// HIGH-PV - Hold if the silo level is too high
IF maxPVEnable AND autoMode THEN
    tonMaxPTrip   (IN := (whiteWaterSiloLevel > maxPVTripEng),       PT := maxPVTripTime);
    tonMaxPRelease(IN := (whiteWaterSiloLevel < maxPVReleaseEng),    PT := maxPVReleaseTime);
    IF tonMaxPTrip.Q    THEN maxPVHoldActive := TRUE;  END_IF;
    IF tonMaxPRelease.Q THEN maxPVHoldActive := FALSE; END_IF;

ELSE
    tonMaxPTrip(IN := FALSE);
    tonMaxPRelease(IN := FALSE);
    maxPVHoldActive := FALSE;
END_IF;

// ============================ PV HOLD aggregation ============================
// NOTE: Requires pvHoldActive : BOOL in VAR section
pvHoldActive := FALSE;
IF autoMode THEN
    pvHoldActive := (minPVEnable AND minPVHoldActive) OR
                    (maxPVEnable AND maxPVHoldActive);
END_IF;


// ============================ Immediate stop / safety/fault =================
IF rStop OR stopCommand THEN
    controlOutputPct := 0.0;
    running := FALSE;
    deviceState := 'Stopping (Stop command)';
    runLatch := FALSE;
    step := 90;
END_IF;

IF vfdFaultFeedback THEN
    deviceState := 'Fault from drive';
    runLatch := FALSE;
    step := 90;
END_IF;

IF NOT allSafetyOK THEN
    deviceState := 'Stopping: safety chain open';
    runLatch := FALSE;
    step := 90;
END_IF;


// ============================ State machine =====================
CASE step OF
    // ------------------------------------------------------------
    0: // Idle
        running := FALSE;
        controlOutputPct := 0.0;
        deviceState := 'Idle';
        vfdStartCmdOut := FALSE;

        // Start request via runLatch (toggled by Start pulse)
        IF runLatch AND NOT stopCommand THEN
            // Safety must be OK; drive must be ready
            // PV hold does NOT block start anymore; it will only inhibit reference to 0%
            IF NOT allSafetyOK THEN
                deviceState := 'Start blocked: safety not OK';
                runLatch := FALSE;
                step := 0;

            ELSIF NOT vfdReady THEN
                deviceState := 'Start blocked: drive not ready';
                runLatch := FALSE;
                step := 0;

            ELSE
                IF pvHoldActive THEN
                    deviceState := 'Starting (PV hold active: output inhibited)';
                ELSE
                    deviceState := 'Starting';
                END_IF;

                vfdStartCmdOut := TRUE;                   // send START to drive
                tonRunFbWait(IN := TRUE, PT := vfdRunFbTimeout);
                step := 10;
            END_IF
        END_IF

    // ------------------------------------------------------------
    10: // Starting (await RUN feedback)
        running := FALSE;
        deviceState := 'Starting (await RUN feedback)';
        vfdStartCmdOut := TRUE;

        // If PV hold is active during start, ensure reference is inhibited to 0%
        IF pvHoldActive THEN
            controlOutputPct := 0.0;
        END_IF;

        // Safety/fault during start => stop
        IF NOT allSafetyOK THEN
            tonRunFbWait(IN := FALSE);
            deviceState := 'Stopping: safety chain open';
            vfdStartCmdOut := FALSE;
            runLatch := FALSE;
            step := 90;

        ELSIF vfdFaultFeedback THEN
            tonRunFbWait(IN := FALSE);
            deviceState := 'Fault from drive';
            vfdStartCmdOut := FALSE;
            runLatch := FALSE;
            step := 90;

        // Interlocks are normal stop only
        ELSIF anyInterlockOpen THEN
            tonRunFbWait(IN := FALSE);
            deviceState := 'Stopping: interlock open';
            vfdStartCmdOut := FALSE;
            runLatch := FALSE;
            step := 90;

        // RUN feedback arrived
        ELSIF vfdRunFeedback THEN
            tonRunFbWait(IN := FALSE);
            step := 20;

        // Timeout
        ELSIF tonRunFbWait.Q THEN
            tonRunFbWait(IN := FALSE);
            deviceState := 'Start failed: RUN feedback timeout';
            vfdStartCmdOut := FALSE;
            runLatch := FALSE;
            step := 90;
        END_IF

    // ------------------------------------------------------------
    20: // Running (control loop)
        running := TRUE;               // may be used to release other devices
        deviceState := 'Running';
        vfdStartCmdOut := TRUE;

        // Supervision
        IF NOT allSafetyOK THEN
            deviceState := 'Stopping: safety chain open';
            vfdStartCmdOut := FALSE;
            runLatch := FALSE;
            step := 90;

        ELSIF vfdFaultFeedback THEN
            deviceState := 'Fault from drive';
            vfdStartCmdOut := FALSE;
            runLatch := FALSE;
            step := 90;

        ELSIF NOT vfdReady THEN
            deviceState := 'Stopping: drive not ready';
            vfdStartCmdOut := FALSE;
            runLatch := FALSE;
            step := 90;

        ELSIF NOT vfdRunFeedback THEN
            deviceState := 'Stopping: RUN feedback lost';
            vfdStartCmdOut := FALSE;
            runLatch := FALSE;
            step := 90;

        // Interlocks → normal stop
        ELSIF anyInterlockOpen THEN
            deviceState := 'Stopping: interlock open';
            vfdStartCmdOut := FALSE;
            runLatch := FALSE;
            step := 90;

        // Start toggled OFF while running => stop
        ELSIF NOT runLatch THEN
            deviceState := 'Stopping (Start toggled off)';
            vfdStartCmdOut := FALSE;
            step := 90;

        ELSE
            // ---- Input filtering (PT1) ----
            IF enableInputFilter THEN
                instPT1(in := whiteWaterSiloLevel, T := inputFilterTime, K := inputFilterGainK, out => pvEngFiltered);
            ELSE
                pvEngFiltered := whiteWaterSiloLevel;
            END_IF

            // ---- Engineering → % scaling ----
            IF enableScaling THEN
                pvPct := _ScaleToPct(pvEngFiltered,       pLoEng, pHiEng);
                spPct := _ScaleToPct(processSetpointAuto, pLoEng, pHiEng);
            ELSE
                pvPct := pvEngFiltered;        // already %
                spPct := processSetpointAuto;  // already %
            END_IF

            // ---- Manual path (HMI) ----
            manualCmd := LIMIT(0.0, processSetpointMan, 100.0);

            // Reverse/direct action by Kp sign
            IF reverseActing THEN
                kpUse := -ABS(kp);
            ELSE
                kpUse :=  ABS(kp);
            END_IF

            // ===================== PV HOLD behavior =====================
            // When PV hold active: keep motor energized, force reference=0.0,
            // and hold PID (avoid error/windup) by forcing SET=ACT and MAN=TRUE.
            IF pvHoldActive THEN

                deviceState := 'Running (PV hold: output inhibited)';
                vfdStartCmdOut := TRUE;        // keep energized
                running := TRUE;               // keep permissives (change to FALSE if you prefer)

                instPID(
                    ACT := pvPct,
                    SET := pvPct,              // hold: SET follows PV -> DIFF ~ 0
                    M_I := 0.0,                // forced output during hold
                    MAN := TRUE,               // hold PID
                    RST := resetPID,
                    KP  := kpUse,
                    TN  := tn,
                    TV  := tv,
//                    LL  := outLowLimitPct,
//                    LH  := outHighLimitPct,
                    Y   => yPID,
                    DIFF=> pidDiff,
                    LIM => pidLimited
                );

                // Output inhibited to zero, motor stays enabled
                controlOutputPct := 0.0;

            ELSE
                // ===================== Normal control =====================
                instPID(
                    ACT := pvPct,
                    SET := spPct,
                    M_I := manualCmd,
                    MAN := NOT autoMode,
                    RST := resetPID,
                    KP  := kpUse,
                    TN  := tn,
                    TV  := tv,
//                    LL  := outLowLimitPct,
//                    LH  := outHighLimitPct,
                    Y   => yPID,
                    DIFF=> pidDiff,
                    LIM => pidLimited
                );

                // Mode select, offset, clamp
                IF autoMode THEN
                    controlOutputPct := yPID;
					instPID.LL := outLowLimitPct;
					instPID.LH := outHighLimitPct;
				
					
                ELSE
                    controlOutputPct := manualCmd;
					instPID.LL := manualCmd;
					instPID.LH := manualCmd;
				
                END_IF

                controlOutputPct := LIMIT(outLowLimitPct, controlOutputPct + outputOffsetPct, outHighLimitPct);
            END_IF
        END_IF

    // ------------------------------------------------------------
    90: // Stopping (normal, de-energize)
        running := FALSE;
        controlOutputPct := 0.0;
        vfdStartCmdOut := FALSE;
        tonRunFbWait(IN := FALSE);

        // Return to Idle once stop released and safety OK
        IF NOT stopCommand AND allSafetyOK THEN
            deviceState := 'Idle';
            step := 0;
        END_IF

    // ------------------------------------------------------------
    ELSE
        running := FALSE;
        controlOutputPct := 0.0;
        deviceState := 'Idle';
        vfdStartCmdOut := FALSE;
        step := 0;
END_CASE;


// =============================== Status code ===============================
IF vfdFaultFeedback THEN
    statusCode := 2;             // Fault
ELSIF running THEN
    statusCode := 1;             // Running
ELSE
    statusCode := 0;             // Idle
END_IF

// HMI feedbacks & status (encapsulates PT1 displays and status code if desired)
_FeedbackDisplay();

// Setpoint input handling (encapsulates TUNE2-based HMI writes & nudges)
_SetpointInputControl();

METHOD _FeedbackDisplay
VAR_INPUT
END_VAR
//instPT1_WhiteWaterSiloDisplay
//whiteWaterLevelDisplay
// 5) HMI DISPLAY SIGNALS (filtered speeds/torques + GROUP status)
instPT1_SpeedDisplay(in := vfdEngFeedback, T := displayFilterTime, K := 1.0, out => vfdEngDisplay);
instPT1_TorqueDisplay (in := vfdTorqueFeedback , T := displayFilterTime, K := 1.0, out => vfdTorqueDisplay);
instPT1_ProcessFeedbackEngDisplay(in := wirePitLevel , T := displayFilterTime, K := 1.0, out => wirePitLevelDisplay);
instPT1_WhiteWaterSiloLevelDisplay(in := whiteWaterSiloLevel , T := displayFilterTime, K := 1.0, out => whiteWaterSiloLevelDisplay);
END_METHOD

// ============================ Helper ============================
METHOD PRIVATE _ScaleToPct : REAL
VAR_INPUT
    xEng  : REAL;  // value in engineering units
    loEng : REAL;  // min eng
    hiEng : REAL;  // max eng
END_VAR
VAR
    span : REAL;
    pct  : REAL;
END_VAR

span := hiEng - loEng;
IF span = 0.0 THEN
    _ScaleToPct := 0.0; // avoid div by zero
ELSE
    pct := (xEng - loEng) / span * 100.0;
    _ScaleToPct := LIMIT(0.0, pct, 100.0);
END_IF
END_METHOD

// ============================================================================
// METHOD: _SetpointInputControl
// Purpose: Handle HMI writes for manual output using OSCAT TUNE2. Any external
//          write to manualOutputPct bigger than the configured step will pulse
//          SET for one scan. No SU/SD buttons here (PressureCtrl doesn’t use them).
// Objetivo: Tratar escrita da HMI no manualOutputPct via TUNE2. Mudança externa
//           > passo gera pulso SET de 1 varredura. Sem botões ↑/↓ neste FB.
// ============================================================================
METHOD PRIVATE _SetpointInputControl
VAR
    spManClamped : REAL;
    spAutoClamped : REAL;
	
END_VAR
// Detect external write (> step): ignore tiny jitter
IF ABS(processSetpointMan - processSetpointManOld) > instTUNE2ManSetpoint.SS THEN
    // Clamp to output limits before writing (garante limites)
    spManClamped := LIMIT(outLowLimitPct, processSetpointMan, outHighLimitPct);

    // One-scan SET pulse into TUNE2 (pulso SET de 1 ciclo)
    instTUNE2ManSetpoint(
        SET_val := spManClamped,
        SET     := TRUE
    );
    instTUNE2ManSetpoint(SET := FALSE);

    // Remember applied value (memoriza)
    processSetpointManOld := processSetpointMan;
ELSE
    // Track last seen to avoid drift (rastreia último observado)
    processSetpointManOld := processSetpointMan;
END_IF;

// Keep TUNE2 active (no SU/SD in this FB)
instTUNE2ManSetpoint(
    SET      := FALSE,
    SU       := processSetpointManInc,
    SD       := processSetpointManDec,
    RST      := FALSE,
    SS       := 0.1,           // step reference (passo de referência)
    FS       := 0.0,                     // unused
    LIMIT_L  := outLowLimitPct,
    LIMIT_H  := outHighLimitPct,
    Y        => processSetpointMan
);




// Detect external write (> step): ignore tiny jitter
IF ABS(processSetpointAuto - processSetpointAutoOld) > instTUNE2AutoSetpoint.SS THEN
    // Clamp to output limits before writing (garante limites)
    spAutoClamped := LIMIT(0, processSetpointAuto, 100);

    // One-scan SET pulse into TUNE2 (pulso SET de 1 ciclo)
    instTUNE2AutoSetpoint(
        SET_val := spAutoClamped,
        SET     := TRUE
    );
    instTUNE2AutoSetpoint(SET := FALSE);

    // Remember applied value (memoriza)
    processSetpointAutoOld := processSetpointAuto;
ELSE
    // Track last seen to avoid drift (rastreia último observado)
    processSetpointAutoOld := processSetpointAuto;
END_IF;

// Keep TUNE2 active (no SU/SD in this FB)
instTUNE2AutoSetpoint(
    SET      := FALSE,
    SU       := processSetpointAutoInc,
    SD       := processSetpointAutoDec,
    RST      := FALSE,
    SS       := 0.1,           // step reference (passo de referência)
    FS       := 0.0,                     // unused
    LIMIT_L  := 0.0,
    LIMIT_H  := 100.0,
    Y        => processSetpointAuto
);
END_METHOD

END_FUNCTION_BLOCK

// ---- Function Blocks/PaperMachine/Auxiliary/FB_ValveProcessControler.TcPOU
(*
    FB_ValveProcessControler (Simplified for Proportional Solenoid)
    Purpose: Generic process controller without VFD sequencing.
             Always evaluates the control loop (equivalent to STEP=20).
             PID (OSCAT CTRL_PID), optional reverse action, PV PT1 filter,
             engineering↔% scaling, low/high PV hold, and HMI displays.

    Status codes: statusCode INT → 0=Inhibited/Idle, 1=Running
*)

FUNCTION_BLOCK FB_ValveProcessControler
VAR_INPUT
    // ===== Manual output & Auto SP nudge =====
    processSetpointManInc        : BOOL;            // Manual output ↑ (0..100%)
    processSetpointManDec        : BOOL;            // Manual output ↓ (0..100%)
    processSetpointManSteps      : REAL := 0.1;

    processSetpointAutoInc       : BOOL;            // Auto SP ↑ (engineering units or %)
    processSetpointAutoDec       : BOOL;            // Auto SP ↓ (engineering units or %)
    processSetpointAutoSteps     : REAL := 1.0;

	holdClosed					: BOOL;				// This should hold the output closed (0.0) while enabled
	
    // ===== Mode =====
    autoMode                     : BOOL;            // TRUE=Automatic / FALSE=Manual
    reverseActing                : BOOL := FALSE;   // TRUE: higher output decreases PV; FALSE: direct

    // ===== Process signals (PV in engineering units) =====
    processFeedbackEng           : REAL;            // PV (engineering units), e.g., bar/kPa/°C/…

    // ===== PID parameters (OSCAT CTRL_PID) =====
    kp                           : REAL := 1.0;     // Proportional gain (sign handled via reverseActing)
    tn                           : REAL := 8.0;     // Integral time [s]
    tv                           : REAL := 0.0;     // Derivative time [s]

    // ===== Output limits & offset =====
    outLowLimitPct               : REAL := 0.0;     // Min output %
    outHighLimitPct              : REAL := 100.0;   // Max output %
    outputOffsetPct              : REAL := 0.0;     // Offset added to final output

    // ===== PID housekeeping =====
    resetPID                     : BOOL;            // Reset integrator

    // ===== Input filter (OSCAT FT_PT1) =====
	deadBand					: REAL := 1.0;
    enableInputFilter            : BOOL := TRUE;    // Enable PV PT1 filter
    inputFilterTime              : TIME := T#300ms; // PT1 time constant
    inputFilterGainK             : REAL := 1.0;     // PT1 gain
    displayFilterTime            : TIME := T#20ms;  // Small PT1 for HMI displays

    // ===== Optional scaling (engineering ↔ %) =====
    enableScaling                : BOOL := TRUE;    // Enable engineering↔% scaling
    pLoEng                       : REAL := 0.0;     // Engineering low bound
    pHiEng                       : REAL := 10.0;    // Engineering high bound

    // ===== Safety (true safety inputs only) =====
    safetyOk                     : BOOL := TRUE;    // Safety chain OK
    estopOk                      : BOOL := TRUE;    // E-Stop loop OK
    guardClosedOk                : BOOL := TRUE;    // Guards/doors closed

    // ===== Interlocks (process permissives) — inhibit output =====
    interlock1                   : BOOL := TRUE;
    interlock2                   : BOOL := TRUE;
    interlock3                   : BOOL := TRUE;
    interlock4                   : BOOL := TRUE;
    interlock5                   : BOOL := TRUE;
    interlock6                   : BOOL := TRUE;

    // ===== Optional low-PV hold =====
    minPVEnable                  : BOOL := FALSE;   // Enable low-PV hold
    minPVTripEng                 : REAL := 0.5;     // Trip threshold (engineering units)
    minPVReleaseEng              : REAL := 0.7;     // Release threshold (engineering units)
    minPVTripTime                : TIME := T#1s;    // PV < trip for this long to trip
    minPVReleaseTime             : TIME := T#1s;    // PV > release for this long to release

    // ===== Optional high-PV hold =====
    maxPVEnable                  : BOOL := FALSE;   // Enable high-PV hold
    maxPVTripEng                 : REAL := 9.5;     // Trip threshold (engineering units)
    maxPVReleaseEng              : REAL := 9.2;     // Release threshold (engineering units)
    maxPVTripTime                : TIME := T#1s;    // PV > trip for this long to trip
    maxPVReleaseTime             : TIME := T#1s;    // PV < release for this long to release
END_VAR

VAR_IN_OUT
    // ===== Exposed setpoints =====
    processSetpointMan           : REAL;            // Manual output 0..100%
    processSetpointAuto          : REAL;            // Auto SP (engineering units or % per configuration)
END_VAR

VAR_OUTPUT
    running                      : BOOL;            // TRUE when permissives OK and no holds
    controlOutputPct             : REAL;            // Final control output 0..100%
    controlOutputPctDisplay             : REAL;            // Final control output 0..100%
	
    pidDiff                      : REAL;            // SET − ACT (post-scaling)
    pidLimited                   : BOOL;            // TRUE if saturated
    deviceState                  : STRING(80);      // Human-readable state

    // ===== Holds =====
    minPVHoldActive              : BOOL;            // Low-PV hold active
    maxPVHoldActive              : BOOL;            // High-PV hold active

    // ===== Status & HMI displays =====
    statusCode                   : INT;             // 0=Inhibited/Idle, 1=Running
    processFeedbackEngDisplay    : REAL;            // PV (engineering units) for HMI
END_VAR

VAR
    // ===== First scan =====
    firstScan                    : BOOL := TRUE;    // TRUE only on first PLC cycle

    // ===== Internals =====
    manualCmd                    : REAL;            // Manual command %
    yPID                         : REAL;            // PID output %
    kpUse                        : REAL;            // Kp adjusted by reverseActing

    // ===== Filtered PV (engineering units) =====
    pvEngFiltered                : REAL;

    // ===== PV & SP in % (post-scaling) =====
    pvPct                        : REAL;
    spPct                        : REAL;

    // ===== Low/High PV timers =====
    tonMinPTrip                  : TON;
    tonMinPRelease               : TON;
    tonMaxPTrip                  : TON;
    tonMaxPRelease               : TON;

    // ===== Instances =====
    instPID                      : CTRL_PID;        // OSCAT PID
    instPT1                      : FT_PT1;          // PV PT1 filter

    // ===== Aggregations =====
    allSafetyOK                  : BOOL := TRUE;            // safetyOk & estopOk & guardClosedOk
    anyInterlockOpen             : BOOL;            // any interlock is FALSE

    // ===== HMI display filters =====
    instPT1_ProcessFeedbackEngDisplay : FT_PT1;     // PT1 for PV display

    // ===== TUNE2 housekeeping =====
    processSetpointManOld        : REAL;            // last observed manual SP
    processSetpointAutoOld       : REAL;            // last observed auto SP
END_VAR

VAR PERSISTENT
    instTUNE2AutoSetpoint        : TUNE2;           // OSCAT TUNE2 for auto SP nudge
    instTUNE2ManSetpoint         : TUNE2;           // OSCAT TUNE2 for manual output
END_VAR

// ============================ Control (STEP 20 equivalent) =====================
// Default safe values
running := FALSE;
controlOutputPct := 0.0;
_SetpointInputControl();

// Inhibit conditions (no start/stop logic — controller is "enabled" only if allowed)
IF NOT allSafetyOK THEN
    deviceState := 'Inhibited: safety chain open';

ELSIF anyInterlockOpen THEN
    deviceState := 'Inhibited: interlock open';

ELSIF holdClosed AND autoMode THEN
    // NEW: force output closed while enabled
    deviceState := 'Held closed';
    running := FALSE;
    controlOutputPct := 0.0;
    controlOutputPctDisplay := 0.0;

    // Optional (recommended): prevent PID windup by forcing MAN=TRUE at 0%
    // Keep scaling/filtering consistent if you need PV/SP for displays; otherwise can omit.
    IF enableInputFilter THEN
        instPT1(in := processFeedbackEng, T := inputFilterTime, K := inputFilterGainK, out => pvEngFiltered);
    ELSE
        pvEngFiltered := processFeedbackEng;
    END_IF

    IF enableScaling THEN
        pvPct := _ScaleToPct(pvEngFiltered,       pLoEng, pHiEng);
        spPct := _ScaleToPct(processSetpointAuto, pLoEng, pHiEng);
    ELSE
        pvPct := pvEngFiltered;
        spPct := processSetpointAuto;
    END_IF

    instPID(
        ACT := pvPct,
        SET := spPct,
        M_I := 0.0,
        MAN := TRUE,
        RST := resetPID, // or TRUE if you prefer to reset integrator while held
        KP  := kpUse,
        TN  := tn,
        TV  := tv,
        SUP := deadBand,
        LL  := 0,
        LH  := 60,
        Y   => yPID,
        DIFF=> pidDiff,
        LIM => pidLimited
    );

ELSIF (minPVEnable AND minPVHoldActive) OR (maxPVEnable AND maxPVHoldActive) THEN
    deviceState := 'Inhibited: PV hold active';

ELSE
    // Allowed to control
    running := TRUE;
    deviceState := 'Running';

    // ---- Input filtering (PT1) ----
    IF enableInputFilter THEN
        instPT1(in := processFeedbackEng, T := inputFilterTime, K := inputFilterGainK, out => pvEngFiltered);
    ELSE
        pvEngFiltered := processFeedbackEng;
    END_IF

    // ---- Engineering → % scaling ----
    IF enableScaling THEN
        pvPct := _ScaleToPct(pvEngFiltered,       pLoEng, pHiEng);
        spPct := _ScaleToPct(processSetpointAuto, pLoEng, pHiEng);
    ELSE
        pvPct := pvEngFiltered;        // already %
        spPct := processSetpointAuto;  // already %
    END_IF

    // ---- Manual path and PID with bumpless transfer ----
    manualCmd := LIMIT(0.0, processSetpointMan, 100.0);

    // Reverse/direct action by Kp sign
    IF reverseActing THEN
        kpUse := -ABS(kp);
    ELSE
        kpUse :=  ABS(kp);
    END_IF

    instPID(
        ACT := pvPct,
        SET := spPct,
        M_I := manualCmd,
        MAN := NOT autoMode,
        RST := resetPID,
        KP  := kpUse,
        TN  := tn,
        TV  := tv,
        SUP := deadBand,
        LL  := 0,
        LH  := 60,
        Y   => yPID,
        DIFF=> pidDiff,
        LIM => pidLimited
    );

    // Mode select, offset, clamp
    IF autoMode THEN
        controlOutputPct := yPID;
    ELSE
        controlOutputPct := manualCmd;
    END_IF
    controlOutputPct := LIMIT(outLowLimitPct, controlOutputPct + outputOffsetPct, outHighLimitPct);
    controlOutputPctDisplay := controlOutputPct;
END_IF;

METHOD _FeedbackDisplay
VAR_INPUT
END_VAR

instPT1_ProcessFeedbackEngDisplay(in := processFeedbackEng , T := displayFilterTime, K := 1.0, out => processFeedbackEngDisplay);
END_METHOD

// ============================ Helper ============================
METHOD PRIVATE _ScaleToPct : REAL
VAR_INPUT
    xEng  : REAL;  // value in engineering units
    loEng : REAL;  // min eng
    hiEng : REAL;  // max eng
END_VAR
VAR
    span : REAL;
    pct  : REAL;
END_VAR

span := hiEng - loEng;
IF span = 0.0 THEN
    _ScaleToPct := 0.0; // avoid div by zero
ELSE
    pct := (xEng - loEng) / span * 100.0;
    _ScaleToPct := LIMIT(0.0, pct, 100.0);
END_IF
END_METHOD

// ============================================================================
// METHOD: _SetpointInputControl
// Purpose: Handle HMI writes for manual output using OSCAT TUNE2. Any external
//          write to manualOutputPct bigger than the configured step will pulse
//          SET for one scan. No SU/SD buttons here (PressureCtrl doesn’t use them).
// Objetivo: Tratar escrita da HMI no manualOutputPct via TUNE2. Mudança externa
//           > passo gera pulso SET de 1 varredura. Sem botões ↑/↓ neste FB.
// ============================================================================
METHOD PRIVATE _SetpointInputControl
VAR
    spManClamped : REAL;
    spAutoClamped : REAL;
	
END_VAR
// Detect external write (> step): ignore tiny jitter
IF ABS(processSetpointMan - processSetpointManOld) > instTUNE2ManSetpoint.SS THEN
    // Clamp to output limits before writing (garante limites)
    spManClamped := LIMIT(outLowLimitPct, processSetpointMan, outHighLimitPct);

    // One-scan SET pulse into TUNE2 (pulso SET de 1 ciclo)
    instTUNE2ManSetpoint(
        SET_val := spManClamped,
        SET     := TRUE
    );
    instTUNE2ManSetpoint(SET := FALSE);

    // Remember applied value (memoriza)
    processSetpointManOld := processSetpointMan;
ELSE
    // Track last seen to avoid drift (rastreia último observado)
    processSetpointManOld := processSetpointMan;
END_IF;

// Keep TUNE2 active (no SU/SD in this FB)
instTUNE2ManSetpoint(
    SET      := FALSE,
    SU       := processSetpointManInc,
    SD       := processSetpointManDec,
    RST      := FALSE,
    SS       := 1.0,           // step reference (passo de referência)
    FS       := 1.0,                     // unused
    LIMIT_L  := outLowLimitPct,
    LIMIT_H  := outHighLimitPct,
    Y        => processSetpointMan
);




// Detect external write (> step): ignore tiny jitter
IF ABS(processSetpointAuto - processSetpointAutoOld) > instTUNE2AutoSetpoint.SS THEN
    // Clamp to output limits before writing (garante limites)
    spAutoClamped := LIMIT(0, processSetpointAuto, 100);

    // One-scan SET pulse into TUNE2 (pulso SET de 1 ciclo)
    instTUNE2AutoSetpoint(
        SET_val := spAutoClamped,
        SET     := TRUE
    );
    instTUNE2AutoSetpoint(SET := FALSE);

    // Remember applied value (memoriza)
    processSetpointAutoOld := processSetpointAuto;
ELSE
    // Track last seen to avoid drift (rastreia último observado)
    processSetpointAutoOld := processSetpointAuto;
END_IF;

// Keep TUNE2 active (no SU/SD in this FB)
instTUNE2AutoSetpoint(
    SET      := FALSE,
    SU       := processSetpointAutoInc,
    SD       := processSetpointAutoDec,
    RST      := FALSE,
    SS       := 0.1,           // step reference (passo de referência)
    FS       := 0.0,                     // unused
    LIMIT_L  := 0,
    LIMIT_H  := 100,
    Y        => processSetpointAuto
);
END_METHOD

END_FUNCTION_BLOCK

// ---- Function Blocks/PaperMachine/DriveControl/FB_DryingSectionDriveControl_V2.TcPOU
FUNCTION_BLOCK FB_DryingSectionDriveControl_V2
VAR_INPUT
    //==============================================================
    // GROUP / INTERLOCKS
    //==============================================================
    startGroup                      : BOOL;  // EN: Start command (pulse / rising edge) / PT: Comando de partida (pulso / borda de subida)
    stopGroup                       : BOOL;  // EN: Stop command (level / maintained) / PT: Comando de parada (nível / mantido)
    groupReset                      : BOOL;  // EN: Reset group faults (HMI / operator reset) / PT: Reset das falhas do grupo (HMI / operador)
    groupNumber                     : INT := 1;   // EN: Group number (1 = first drying group / 2 = second...) / PT: Número do grupo (1 = 1º grupo de secagem / 2 = 2º ...)

    //==============================================================
    // DRIVE STATUS INPUTS (VFDs) — UPPER GROUP
    //==============================================================
    upperMasterReady                : BOOL;  // EN: Upper master ready (no trip) = TRUE / PT: Mestre superior pronto (sem trip) = TRUE
    upperMasterVfdRunFeedback       : BOOL;  // EN: Upper master RUN feedback = running / PT: Retorno de RUN do mestre superior = rodando
    upperMasterVfdFaultFeedback     : BOOL;  // EN: Upper master fault/alarm = TRUE when drive has fault / PT: Falha/alarme do mestre superior = TRUE quando drive falhar
    upperSlave1VfdReady             : BOOL;  // EN: Upper slave 1 ready / PT: Escravo 1 superior pronto
    upperSlave1VfdRunFeedback       : BOOL;  // EN: Upper slave 1 RUN feedback / PT: Retorno de RUN do escravo 1 superior
    upperSlave1VfdFaultFeedback     : BOOL;  // EN: Upper slave 1 fault/alarm / PT: Falha/alarme do escravo 1 superior
    upperSlave2VfdReady             : BOOL;  // EN: Upper slave 2 ready / PT: Escravo 2 superior pronto
    upperSlave2VfdRunFeedback       : BOOL;  // EN: Upper slave 2 RUN feedback / PT: Retorno de RUN do escravo 2 superior
    upperSlave2VfdFaultFeedback     : BOOL;  // EN: Upper slave 2 fault/alarm / PT: Falha/alarme do escravo 2 superior

    //==============================================================
    // DRIVE STATUS INPUTS (VFDs) — LOWER GROUP
    //==============================================================
    lowerMasterReady                : BOOL;  // EN: Lower master ready (no trip) = TRUE / PT: Mestre inferior pronto (sem trip) = TRUE
    lowerMasterVfdRunFeedback       : BOOL;  // EN: Lower master RUN feedback / PT: Retorno de RUN do mestre inferior
    lowerMasterVfdFaultFeedback     : BOOL;  // EN: Lower master fault/alarm / PT: Falha/alarme do mestre inferior
    lowerSlave1VfdReady             : BOOL;  // EN: Lower slave 1 ready / PT: Escravo 1 inferior pronto
    lowerSlave1VfdRunFeedback       : BOOL;  // EN: Lower slave 1 RUN feedback / PT: Retorno de RUN do escravo 1 inferior
    lowerSlave1VfdFaultFeedback     : BOOL;  // EN: Lower slave 1 fault/alarm / PT: Falha/alarme do escravo 1 inferior
    lowerSlave2VfdReady             : BOOL;  // EN: Lower slave 2 ready / PT: Escravo 2 inferior pronto
    lowerSlave2VfdRunFeedback       : BOOL;  // EN: Lower slave 2 RUN feedback / PT: Retorno de RUN do escravo 2 inferior
    lowerSlave2VfdFaultFeedback     : BOOL;  // EN: Lower slave 2 fault/alarm / PT: Falha/alarme do escravo 2 inferior

    //==============================================================
    // DRYING SECTION — COOLING MOTOR FAULTS (PER DRIVE)
    //==============================================================
    upperMasterCoolingMotorFault    : BOOL;  // EN: Cooling motor fault for upper master / PT: Falha do motor de ventilação do mestre superior
    upperSlave1CoolingMotorFault    : BOOL;  // EN: Cooling motor fault for upper slave 1 / PT: Falha do motor de ventilação do escravo 1 superior
    upperSlave2CoolingMotorFault    : BOOL;  // EN: Cooling motor fault for upper slave 2 / PT: Falha do motor de ventilação do escravo 2 superior

    lowerMasterCoolingMotorFault    : BOOL;  // EN: Cooling motor fault for lower master / PT: Falha do motor de ventilação do mestre inferior
    lowerSlave1CoolingMotorFault    : BOOL;  // EN: Cooling motor fault for lower slave 1 / PT: Falha do motor de ventilação do escravo 1 inferior
    lowerSlave2CoolingMotorFault    : BOOL;  // EN: Cooling motor fault for lower slave 2 / PT: Falha do motor de ventilação do escravo 2 inferior

    //==============================================================
    // FABRIC / WIRE STRETCHERS (ACTUATORS)
    //==============================================================
    upperDryingSectionFabricStretcherMotorFault : BOOL;  // EN: Upper fabric/wire stretcher motor fault / PT: Falha no motor de estiramento da tela superior
    lowerDryingSectionFabricStretcherMotorFault : BOOL;  // EN: Lower fabric/wire stretcher motor fault / PT: Falha no motor de estiramento da tela inferior

    upperDryingSectionFabricStretchCmd     : BOOL;  // EN: Command to stretch upper fabric / PT: Comando para esticar a tela superior
    upperDryingSectionFabricUnstretchCmd   : BOOL;  // EN: Command to unstretch upper fabric / PT: Comando para afrouxar a tela superior
    lowerDryingSectionFabricStretchCmd     : BOOL;  // EN: Command to stretch lower fabric / PT: Comando para esticar a tela inferior
    lowerDryingSectionFabricUnstretchCmd   : BOOL;  // EN: Command to unstretch lower fabric / PT: Comando para afrouxar a tela inferior

    //==============================================================
    // FABRIC / WIRE OVERRUN SENSORS
    //==============================================================
    upperDryingSectionFabricOverrunOperatorSideSensor : BOOL;  // EN: Upper fabric overrun sensor — operator side / PT: Sensor de sobrecurso da tela superior — lado operador
    upperDryingSectionFabricOverrunDriveSideSensor    : BOOL;  // EN: Upper fabric overrun sensor — drive side / PT: Sensor de sobrecurso da tela superior — lado acionamento
    lowerDryingSectionFabricOverrunOperatorSideSensor : BOOL;  // EN: Lower fabric overrun sensor — operator side / PT: Sensor de sobrecurso da tela inferior — lado operador
    lowerDryingSectionFabricOverrunDriveSideSensor    : BOOL;  // EN: Lower fabric overrun sensor — drive side / PT: Sensor de sobrecurso da tela inferior — lado acionamento

    //────────────────────────────────────────────
    // PICK-UP ROLL POSITIONER / POSICIONADOR DO ROLO PICK-UP
    //────────────────────────────────────────────
    pickUpRollPosCmdFwd              : BOOL; // EN: Command to move pick-up roll forward / PT: Comando para avançar o rolo pick-up
    pickUpRollPosCmdRev              : BOOL; // EN: Command to move pick-up roll reverse / PT: Comando para recuar o rolo pick-up
    pickUpRollPosFault               : BOOL; // EN: Positioner fault (hydraulic/pneumatic/electric) / PT: Falha no atuador de posicionamento
    pickUpRollPosLimitFwd            : BOOL; // EN: Forward end-limit switch / PT: Fim de curso frontal
    pickUpRollPosLimitRev            : BOOL; // EN: Reverse end-limit switch / PT: Fim de curso traseiro

    //────────────────────────────────────────────
    // BABYDRYER SCRAPER OSCILLATOR
    //────────────────────────────────────────────
    babyDryerScraperOscCmd           : BOOL; // EN: Start baby dryer scraper oscillation / PT: Comando de partida da oscilação da raspa do babydryer
    babyDryerScraperOscFault         : BOOL; // EN: Baby dryer scraper oscillator fault / PT: Falha no oscilador da raspa do babydryer
    babyDryerScraperOscRunning       : BOOL; // EN: Baby dryer scraper oscillator running / PT: Oscilador da raspa do babydryer em movimento

    //────────────────────────────────────────────
    // UPPER GROUP SCRAPER OSCILLATOR
    //────────────────────────────────────────────
    upperGroupScraperOscCmd          : BOOL; // EN: Start upper group scraper oscillation / PT: Comando de oscilação da raspa do grupo superior
    upperGroupScraperOscFault        : BOOL; // EN: Upper group scraper oscillator fault / PT: Falha no oscilador da raspa do grupo superior
    upperGroupScraperOscRunning      : BOOL; // EN: Upper group scraper oscillator running / PT: Oscilador da raspa do grupo superior em movimento

    //────────────────────────────────────────────
    // LOWER GROUP SCRAPER OSCILLATOR
    //────────────────────────────────────────────
    lowerGroupScraperOscCmd          : BOOL; // EN: Start lower group scraper oscillation / PT: Comando de oscilação da raspa do grupo inferior
    lowerGroupScraperOscFault        : BOOL; // EN: Lower group scraper oscillator fault / PT: Falha no oscilador da raspa do grupo inferior
    lowerGroupScraperOscRunning      : BOOL; // EN: Lower group scraper oscillator running / PT: Oscilador da raspa do grupo inferior em movimento

    //==============================================================
    // SPEED SETPOINTS / MODE
    //==============================================================
    groupAutoSpeedMPM                : REAL;  // EN: Auto speed setpoint [m/min] / PT: Setpoint de velocidade em automático [m/min]
    groupManualSpeedMPM              : REAL := 50.0;   // EN: Manual speed reference [m/min] / PT: Velocidade em manual [m/min]
    groupMasterMaxSpeedRPM                    : REAL := 750.0;  //Velocidade maxima do motor em RPM
    groupSpeedAutoMan                : BOOL;           // EN: 0 = Manual, 1 = Auto / PT: 0 = Manual, 1 = Automático

    //==============================================================
    // FEEDBACKS (FROM DRIVES / SENSORS)
    //==============================================================
    // Upper group
    upperMasterSpeedFeedback         : REAL;  // EN: Upper master speed feedback [m/min or %] / PT: Retorno de velocidade do mestre superior [m/min ou %]
    upperMasterTorqueFeedback        : REAL;  // EN: Upper master torque feedback [% or Nm] / PT: Retorno de torque do mestre superior [% ou Nm]
    upperSlave1SpeedFeedback         : REAL;  // EN: Upper slave 1 speed feedback / PT: Retorno de velocidade do escravo 1 superior
    upperSlave1TorqueFeedback        : REAL;  // EN: Upper slave 1 torque feedback / PT: Retorno de torque do escravo 1 superior
    upperSlave2SpeedFeedback         : REAL;  // EN: Upper slave 2 speed feedback / PT: Retorno de velocidade do escravo 2 superior
    upperSlave2TorqueFeedback        : REAL;  // EN: Upper slave 2 torque feedback / PT: Retorno de torque do escravo 2 superior

    // Lower group
    lowerMasterSpeedFeedback         : REAL;  // EN: Lower master speed feedback / PT: Retorno de velocidade do mestre inferior
    lowerMasterTorqueFeedback        : REAL;  // EN: Lower master torque feedback / PT: Retorno de torque do mestre inferior
    lowerSlave1SpeedFeedback         : REAL;  // EN: Lower slave 1 speed feedback / PT: Retorno de velocidade do escravo 1 inferior
    lowerSlave1TorqueFeedback        : REAL;  // EN: Lower slave 1 torque feedback / PT: Retorno de torque do escravo 1 inferior
    lowerSlave2SpeedFeedback         : REAL;  // EN: Lower slave 2 speed feedback / PT: Retorno de velocidade do escravo 2 inferior
    lowerSlave2TorqueFeedback        : REAL;  // EN: Lower slave 2 torque feedback / PT: Retorno de torque do escravo 2 inferior

    //==============================================================
    // RATIO / OFFSETS (FOLLOWING / TRIM LOGIC)
    //==============================================================
    masterSlaveGearRatio             : REAL := 1.0;   // EN: Slave/master speed ratio (XXX: "diference" in original) / PT: Relação de velocidade escravo/mestre (XXX: "diference" no original)
    interGroupGearRatio              : REAL := 1.0;   // EN: Speed ratio between groups / PT: Relação de velocidade entre grupos
    slaveTorqueOfsset                : REAL := 0.0;   // EN: XXX: "Ofsset" → torque trim offset applied to slaves [% or Nm] / PT: XXX: "Ofsset" → offset de torque aplicado aos escravos [% ou Nm]
    slaveSpeedOffset                 : REAL := 10.0;  // EN: Speed offset between master and slaves [% of master] / PT: Offset de velocidade entre mestre e escravos [% do mestre]
    upperAndLowerSpeedOffset         : REAL := 1.0;   // EN: XXX: "uper" → Speed offset between upper and lower groups [%] / PT: XXX: "uper" → Offset de velocidade entre grupo superior e inferior [%]

    groupRecoverSpeedCmd             : BOOL;          // EN: Command to temporarily recover group speed / PT: Comando para recuperar temporariamente a velocidade do grupo
    groupRecoverIncrement            : REAL := 5.0;   // EN: Recovery speed increment [m/min or %] / PT: Incremento de recuperação de velocidade [m/min ou %]

    groupSpeedDifInc                 : BOOL;          // EN: Increment group-to-group speed difference / PT: Incrementa diferença de velocidade entre grupos
    groupSpeedDifDec                 : BOOL;          // EN: Decrement group-to-group speed difference / PT: Decrementa diferença de velocidade entre grupos
    groupSpeedDifLimHigh             : REAL := 20.0;  // EN: Upper limit for group speed difference [%] / PT: Limite superior da diferença de velocidade entre grupos [%]
    groupSpeedDifLimLow              : REAL := -20.0; // EN: Lower limit for group speed difference [%] / PT: Limite inferior da diferença de velocidade entre grupos [%]

    //==============================================================
    // TORQUE CONTROL / LIMITS
    //==============================================================
    enableTorquePid                  : BOOL := FALSE; // EN: Enable torque trim PID (OSCAT) / PT: Habilita o PID de trim de torque (OSCAT)
    torqueTrimLimit                  : REAL := 10.0;  // EN: Max magnitude for torque trim (|trim| ≤ value) / PT: Limite máximo para o trim de torque (|trim| ≤ valor)
    torqueLimitMinPct                : REAL := 0.0;   // EN: Min torque limit for slaves [%] / PT: Limite mínimo de torque para escravos [%]
    torqueLimitMaxPct                : REAL := 150.0; // EN: Max torque limit for slaves [%] / PT: Limite máximo de torque para escravos [%]
    torqueDeadbandPct                : REAL := 1.0;   // EN: Deadband for torque error [%] / PT: Banda morta para erro de torque [%]
    torqueFilterTime                 : TIME := T#5MS; // EN: Time constant for torque measurement filter / PT: Constante de tempo do filtro da medição de torque
    displayFilterTime                : TIME := T#20ms;// EN: Time constant for HMI display filter / PT: Constante de tempo do filtro de exibição para HMI

    //----- OSCAT CTRL_PID parameters (torque trim) -----
    torqueCtrlKp                     : REAL := 1.0;   // EN: Proportional gain / PT: Ganho proporcional
    torqueCtrlTn                     : REAL := 8.0;   // EN: Integral time [s] / PT: Tempo integral [s]
    torqueCtrlTv                     : REAL := 0.0;   // EN: Derivative time [s] / PT: Tempo derivativo [s]

    //==============================================================
    // DYNAMICS / LIMITS
    //==============================================================
    rampRate                         : REAL := 0.01;  // EN: Reference acceleration rate for ramp block [%/s] / PT: Taxa de aceleração da rampa de referência [%/s]
    speedDiferenceLimit              : REAL := 5.0;   // EN: XXX: "Diference" → Max allowed speed difference between groups/slaves [%] / PT: XXX: "Diference" → Diferença máx. de velocidade permitida entre grupos/escravos [%]


	
	steamPressureAutoMan				: BOOL;
	steamPressureAutoSetpoint			: REAL;
	steamPressureManualSetpoint			: REAL;
	steamPressureFeedback				: REAL;

	steamPressureKp : REAL := 1.0;  // PID Kp for Group 1 steam pressure
	steamPressureTn : REAL := 8.0;  // PID Tn for Group 1 steam pressure
	steamPressureTv : REAL := 0.0;  // PID Tv for Group 1 steam pressure	
	
    //==============================================================
    // ROLL DIAMETERS
    //==============================================================	
	upperMasterDiameter	: REAL;
	upperSlave1Diameter	: REAL;
	upperSlave2Diameter	: REAL;

	lowerMasterDiameter	: REAL;
	lowerSlave1Diameter	: REAL;
	lowerSlave2Diameter	: REAL;
	
	
END_VAR


VAR_OUTPUT
    //==============================================================
    // STATE / DIAGNOSTICS
    //==============================================================
    deviceState                      : STRING;        // EN: Current human-readable device/group state / PT: Estado atual do dispositivo/grupo (texto)
    groupFault                       : BOOL;          // EN: Group fault present (interlock) / PT: Falha do grupo presente (intertravamento)

    statusCode                       : INT;           // EN: 0=Idle, 1=Starting, 2=Running, 3=Fault / PT: 0=Parado, 1=Partindo, 2=Rodando, 3=Falha
    currentSpeedDifence              : REAL;          // EN: XXX: "Difence" → Current group-to-group speed difference [%] / PT: XXX: "Difence" → Diferença de velocidade atual entre grupos [%]
    groupSpeedOffset                 : REAL := 0.0;   // EN: Current group speed offset vs previous group [%] / PT: Offset de velocidade atual do grupo em relação ao grupo anterior [%]

    //==============================================================
    // SPEED REFERENCES (TO DRIVES) — 0..100%
    //==============================================================
    upperMasterDriveSpeedRefRPM      : REAL;  // EN: Speed reference for upper master drive [%] / PT: Referência de velocidade para o drive mestre superior [%]
    upperSlave1DriveSpeedRefRPM      : REAL;  // EN: Speed reference for upper slave 1 [%] / PT: Referência de velocidade para o drive escravo 1 superior [%]
    upperSlave2DriveSpeedRefRPM      : REAL;  // EN: Speed reference for upper slave 2 [%] / PT: Referência de velocidade para o drive escravo 2 superior [%]
  
	  lowerMasterDriveSpeedRefRPM      : REAL;  // EN: Speed reference for lower master [%] / PT: Referência de velocidade para o drive mestre inferior [%]
    lowerSlave1DriveSpeedRefRPM      : REAL;  // EN: Speed reference for lower slave 1 [%] / PT: Referência de velocidade para o drive escravo 1 inferior [%]
    lowerSlave2DriveSpeedRefRPM      : REAL;  // EN: Speed reference for lower slave 2 [%] / PT: Referência de velocidade para o drive escravo 2 inferior [%]



    nextGroupSpeedRefRPM             : REAL;  // EN: Suggested speed ref for next downstream group [%] / PT: Velocidade sugerida para o próximo grupo à jusante [%]
    nextGroupSpeedRefMPM             : REAL;  // EN: Suggested speed ref for next downstream group [m/min] / PT: Velocidade sugerida para o próximo grupo à jusante [m/min]

    //==============================================================
    // TORQUE REFERENCES / LIMITS (TO SLAVE DRIVES)
    //==============================================================
    upperSlave1DriveTorqueRefPct     : REAL;  // EN: Torque reference for upper slave 1 [% or Nm] / PT: Referência de torque para o escravo 1 superior [% ou Nm]
    upperSlave2DriveTorqueRefPct     : REAL;  // EN: Torque reference for upper slave 2 [% or Nm] / PT: Referência de torque para o escravo 2 superior [% ou Nm]
    lowerSlave1DriveTorqueRefPct     : REAL;  // EN: Torque reference for lower slave 1 [% or Nm] / PT: Referência de torque para o escravo 1 inferior [% ou Nm]
    lowerSlave2DriveTorqueRefPct     : REAL;  // EN: Torque reference for lower slave 2 [% or Nm] / PT: Referência de torque para o escravo 2 inferior [% ou Nm]
    slaveDriveTorqueLimit            : REAL;  // EN: Common torque limit applied to all slave drives [% or Nm] / PT: Limite de torque comum aplicado a todos os drives escravos [% ou Nm]

    //==============================================================
    // DRIVE COMMANDS (ENABLE / RESET)
    //==============================================================
    upperMasterDriveEnable           : BOOL;  // EN: Enable cmd to upper master drive / PT: Comando de habilitar para o drive mestre superior
    upperMasterDriveReset            : BOOL;  // EN: Reset cmd (pulse) to clear upper master fault / PT: Comando de reset (pulso) para limpar falha do mestre superior
    upperSlave1DriveEnable           : BOOL;  // EN: Enable cmd to upper slave 1 / PT: Comando de habilitar para o escravo 1 superior
    upperSlave1DriveReset            : BOOL;  // EN: Reset cmd to upper slave 1 / PT: Comando de reset para o escravo 1 superior
    upperSlave2DriveEnable           : BOOL;  // EN: Enable cmd to upper slave 2 / PT: Comando de habilitar para o escravo 2 superior
    upperSlave2DriveReset            : BOOL;  // EN: Reset cmd to upper slave 2 / PT: Comando de reset para o escravo 2 superior

    lowerMasterDriveEnable           : BOOL;  // EN: Enable cmd to lower master / PT: Comando de habilitar para o mestre inferior
    lowerMasterDriveReset            : BOOL;  // EN: Reset cmd to lower master / PT: Comando de reset para o mestre inferior
    lowerSlave1DriveEnable           : BOOL;  // EN: Enable cmd to lower slave 1 / PT: Comando de habilitar para o escravo 1 inferior
    lowerSlave1DriveReset            : BOOL;  // EN: Reset cmd to lower slave 1 / PT: Comando de reset para o escravo 1 inferior
    lowerSlave2DriveEnable           : BOOL;  // EN: Enable cmd to lower slave 2 / PT: Comando de habilitar para o escravo 2 inferior
    lowerSlave2DriveReset            : BOOL;  // EN: Reset cmd to lower slave 2 / PT: Comando de reset para o escravo 2 inferior

    //==============================================================
    // HMI — FILTERED DISPLAYS
    //==============================================================

    upperMasterTorqueFilteredDisplay   : REAL; // EN: Filtered upper master torque for HMI / PT: Torque filtrado do mestre superior para HMI
    upperSlave1TorqueFilteredDisplay   : REAL; // EN: Filtered upper slave 1 torque for HMI / PT: Torque filtrado do escravo 1 superior para HMI
    upperSlave2TorqueFilteredDisplay   : REAL; // EN: Filtered upper slave 2 torque for HMI / PT: Torque filtrado do escravo 2 superior para HMI
    lowerMasterTorqueFilteredDisplay   : REAL; // EN: Filtered lower master torque for HMI / PT: Torque filtrado do mestre inferior para HMI
    lowerSlave1TorqueFilteredDisplay   : REAL; // EN: Filtered lower slave 1 torque for HMI / PT: Torque filtrado do escravo 1 inferior para HMI
    lowerSlave2TorqueFilteredDisplay   : REAL; // EN: Filtered lower slave 2 torque for HMI / PT: Torque filtrado do escravo 2 inferior para HMI

    //==============================================================
    // PER-DRIVE STATUS CODES (HMI)
    //==============================================================
    upperMasterStatusCode            : INT;  // EN: Upper master status (0=Idle,1=Start,2=Run,3=Fault) / PT: Status do mestre superior (0=Parado,1=Partida,2=Rodando,3=Falha)
    upperSlave1StatusCode            : INT;  // EN: Upper slave 1 status / PT: Status do escravo 1 superior
    upperSlave2StatusCode            : INT;  // EN: Upper slave 2 status / PT: Status do escravo 2 superior
    lowerMasterStatusCode            : INT;  // EN: Lower master status / PT: Status do mestre inferior
    lowerSlave1StatusCode            : INT;  // EN: Lower slave 1 status / PT: Status do escravo 1 inferior
    lowerSlave2StatusCode            : INT;  // EN: Lower slave 2 status / PT: Status do escravo 2 inferior

    //==============================================================
    // FABRIC / WIRE STRETCHER OUTPUTS
    //==============================================================
    upperDryingSectionFabricStretch   : BOOL; // EN: Output to stretch upper fabric (actuator ON fwd) / PT: Saída para esticar a tela superior (acionar atuador para frente)
    upperDryingSectionFabricUnstretch : BOOL; // EN: Output to unstretch upper fabric (actuator ON rev) / PT: Saída para afrouxar a tela superior (acionar atuador para trás)
    lowerDryingSectionFabricStretch   : BOOL; // EN: Output to stretch lower fabric / PT: Saída para esticar a tela inferior
    lowerDryingSectionFabricUnstretch : BOOL; // EN: Output to unstretch lower fabric / PT: Saída para afrouxar a tela inferior

    //────────────────────────────────────────────
    // PICK-UP ROLL POSITIONER / POSICIONADOR DO ROLO PICK-UP
    //────────────────────────────────────────────
    pickUpRollPosRunFwd               : BOOL; // EN: Run pick-up positioner forward / PT: Acionar posicionador do pick-up para frente
    pickUpRollPosRunRev               : BOOL; // EN: Run pick-up positioner reverse / PT: Acionar posicionador do pick-up para trás

    //────────────────────────────────────────────
    // BABYDRYER SCRAPER OSCILLATOR / OSCILADOR DA RASPA BABYDRYER
    //────────────────────────────────────────────
    babyDryerScraperOscRun            : BOOL; // EN: Activate baby dryer scraper oscillator / PT: Acionar oscilador da raspa do babydryer

    //────────────────────────────────────────────
    // UPPER GROUP SCRAPER OSCILLATOR / OSCILADOR DA RASPA GRUPO SUPERIOR
    //────────────────────────────────────────────
    upperGroupScraperOscRun           : BOOL; // EN: Activate upper group scraper oscillator / PT: Acionar oscilador da raspa do grupo superior

    //────────────────────────────────────────────
    // LOWER GROUP SCRAPER OSCILLATOR / OSCILADOR DA RASPA GRUPO INFERIOR
    //────────────────────────────────────────────
    lowerGroupScraperOscRun           : BOOL; // EN: Activate lower group scraper oscillator / PT: Acionar oscilador da raspa do grupo inferior

   

	steamPressureControllerOutput		: REAL;


    upperMasterSpeedMPM : REAL;
    upperSlave1SpeedMPM : REAL;
    upperSlave2SpeedMPM : REAL;
    lowerMasterSpeedMPM : REAL;
    lowerSlave1SpeedMPM : REAL;
    lowerSlave2SpeedMPM : REAL;	

    upperMasterSpeedRPM : REAL;
    upperSlave1SpeedRPM : REAL;
    upperSlave2SpeedRPM : REAL;
    lowerMasterSpeedRPM : REAL;
    lowerSlave1SpeedRPM : REAL;
    lowerSlave2SpeedRPM : REAL;		
	
	 //==============================================================
    // HMI ALARMS STRUCT
    //==============================================================
    hmiAlarms                          : PaperMachine_TypeHmiAlarms;  // EN: HMI alarms structure for drying section / PT: Estrutura de alarmes da HMI para a seção de secagem
END_VAR


VAR
    //==============================================================
    // INTERNAL — STATE / EDGE DETECTION
    //==============================================================
    state                           : INT;   // EN: Internal state (0=IDLE,1=ENABLE,2=WAIT_EN,3=RAMP_EN,4=RUN,5=STOPPING,10=FAULT) / PT: Estado interno (0=IDLE,1=HABILITA,2=ESPERA_HAB,3=RAMPA,4=RODANDO,5=PARANDO,10=FALHA)
    startGroupOld                   : BOOL;  // EN: Previous cycle value of startGroup / PT: Valor do ciclo anterior de startGroup
    stopGroupOld                    : BOOL;  // EN: Previous cycle value of stopGroup / PT: Valor do ciclo anterior de stopGroup
    rStart                          : BOOL;  // EN: Rising edge of startGroup / PT: Borda de subida do startGroup
    rStop                           : BOOL;  // EN: Rising edge of stopGroup / PT: Borda de subida do stopGroup

    //==============================================================
    // INTERNAL — RAMP / REFERENCE SHAPING
    //==============================================================
    rampTargetRPM                   : REAL;        // EN: Target reference for S-ramp [0..100%] / PT: Referência alvo para a rampa S [0..100%]
    instFB_Gen_SRamp                : FB_Gen_SRamp;// EN: S-ramp block instance / PT: Instância do bloco de rampa S
    rampReset                       : BOOL;        // EN: Reset ramp (force output to 0) / PT: Resetar rampa (força saída para 0)
    useRamp                         : BOOL;        // EN: TRUE = apply ramp, FALSE = direct feed-through / PT: TRUE = aplica rampa, FALSE = passa direto

    //==============================================================
    // INTERNAL — TIMERS / THRESHOLDS
    //==============================================================
    instTONEnableWait               : TON;         // EN: Timer to wait drives ready / PT: Temporizador para aguardar drives prontos
    instTONStopWait                 : TON;         // EN: Timer to wait drives stop / PT: Temporizador para aguardar parada dos drives
    enableTimeout                   : TIME := T#5s;// EN: Max allowed time to get ready / PT: Tempo máximo para habilitar
    stopTimeout                     : TIME := T#8s;// EN: Max allowed time to stop / PT: Tempo máximo para parar
    speedZeroThresholdPct           : REAL := 4.0; // EN: Consider speed = 0 when reference ≤ this [%] / PT: Considera velocidade = 0 quando referência ≤ este valor [%]
    epsRefPct                       : REAL := 0.05;// EN: Small epsilon to avoid chattering / PT: Pequeno epsilon para evitar oscilações

    //==============================================================
    // INTERNAL — TORQUE FILTERING
    //==============================================================
    torqueFiltY                     : REAL;        // EN: Internal filtered torque value / PT: Valor interno de torque filtrado
    torqueFiltInit                  : BOOL;        // EN: One-shot flag to init filter / PT: Flag de um ciclo para iniciar o filtro
    instsFT_PT1UpperTorqueFilter    : FT_PT1;      // EN: PT1 filter for upper group torque / PT: Filtro PT1 para torque do grupo superior
    instsFT_PT1LowerTorqueFilter    : FT_PT1;      // EN: PT1 filter for lower group torque / PT: Filtro PT1 para torque do grupo inferior

    //==============================================================
    // INTERNAL — SUPERVISION
    //==============================================================
    instTONSpeedDifDelay            : TON;         // EN: Delay before raising speed-difference alarm / PT: Atraso antes de levantar alarme de diferença de velocidade

    //==============================================================
    // HMI FILTERS — PT1 (DISPLAY ONLY)
    //==============================================================
    instPT1_UpperMasterSpeedDisplay : FT_PT1;      // EN: Display filter for upper master speed / PT: Filtro de exibição para velocidade do mestre superior
    instPT1_UpperMasterTorqueDisplay: FT_PT1;      // EN: Display filter for upper master torque / PT: Filtro de exibição para torque do mestre superior
    instPT1_UpperSlave1SpeedDisplay : FT_PT1;      // EN: Display filter for upper slave 1 speed / PT: Filtro de exibição para velocidade do escravo 1 superior
    instPT1_UpperSlave1TorqueDisplay: FT_PT1;      // EN: Display filter for upper slave 1 torque / PT: Filtro de exibição para torque do escravo 1 superior
    instPT1_UpperSlave2SpeedDisplay : FT_PT1;      // EN: Display filter for upper slave 2 speed / PT: Filtro de exibição para velocidade do escravo 2 superior
    instPT1_UpperSlave2TorqueDisplay: FT_PT1;      // EN: Display filter for upper slave 2 torque / PT: Filtro de exibição para torque do escravo 2 superior
    instPT1_LowerMasterSpeedDisplay : FT_PT1;      // EN: Display filter for lower master speed / PT: Filtro de exibição para velocidade do mestre inferior
    instPT1_LowerMasterTorqueDisplay: FT_PT1;      // EN: Display filter for lower master torque / PT: Filtro de exibição para torque do mestre inferior
    instPT1_LowerSlave1SpeedDisplay : FT_PT1;      // EN: Display filter for lower slave 1 speed / PT: Filtro de exibição para velocidade do escravo 1 inferior
    instPT1_LowerSlave1TorqueDisplay: FT_PT1;      // EN: Display filter for lower slave 1 torque / PT: Filtro de exibição para torque do escravo 1 inferior
    instPT1_LowerSlave2SpeedDisplay : FT_PT1;      // EN: Display filter for lower slave 2 speed / PT: Filtro de exibição para velocidade do escravo 2 inferior
    instPT1_LowerSlave2TorqueDisplay: FT_PT1;      // EN: Display filter for lower slave 2 torque / PT: Filtro de exibição para torque do escravo 2 inferior

    //==============================================================
    // INTERNAL — TORQUE TRIM PID (OSCAT CTRL_PID)
    //==============================================================
    instCTRL_PID_UpperTorqueTrim    : CTRL_PID;    // EN: PID instance for upper group torque trim / PT: Instância PID para trim de torque do grupo superior
    instCTRL_PID_LowerTorqueTrim    : CTRL_PID;    // EN: PID instance for lower group torque trim / PT: Instância PID para trim de torque do grupo inferior

    instCTRL_PID_TemperatureController    : CTRL_PID;    
	
	
	upperMasterSpeedFilteredFeedback : REAL; // EN: Filtered upper master speed for HMI [m/min] / PT: Velocidade filtrada do mestre superior para HMI [m/min]
    upperSlave1SpeedFilteredFeedback : REAL; // EN: Filtered upper slave 1 speed for HMI [m/min] / PT: Velocidade filtrada do escravo 1 superior para HMI [m/min]
    upperSlave2SpeedFilteredFeedback : REAL; // EN: Filtered upper slave 2 speed for HMI [m/min] / PT: Velocidade filtrada do escravo 2 superior para HMI [m/min]
    lowerMasterSpeedFilteredFeedback : REAL; // EN: Filtered lower master speed for HMI [m/min] / PT: Velocidade filtrada do mestre inferior para HMI [m/min]
    lowerSlave1SpeedFilteredFeedback : REAL; // EN: Filtered lower slave 1 speed for HMI [m/min] / PT: Velocidade filtrada do escravo 1 inferior para HMI [m/min]
    lowerSlave2SpeedFilteredFeedback : REAL; // EN: Filtered lower slave 2 speed for HMI [m/min] / PT: Velocidade filtrada do escravo 2 inferior para HMI [m/min]

	// Upper group (surface speed setpoints in m/min)
	upperMasterSpeedSetpointMPM : REAL;
	upperSlave1SpeedSetpointMPM : REAL;
	upperSlave2SpeedSetpointMPM : REAL;
	
	// Lower group (surface speed setpoints in m/min)
	lowerMasterSpeedSetpointMPM : REAL;
	lowerSlave1SpeedSetpointMPM : REAL;
	lowerSlave2SpeedSetpointMPM : REAL;
		
    // Upper group gear ratios (reference: upper master)
    upperToLowerMasterRatio    : REAL;
    upperToUpperSlave1Ratio    : REAL;
    upperToUpperSlave2Ratio    : REAL;

    // Lower group gear ratios (reference: lower master)
    lowerToUpperMasterRatio    : REAL;
    lowerToLowerSlave1Ratio    : REAL;
    lowerToLowerSlave2Ratio    : REAL;	
	
	
	masterMaxSpeedMPM: REAL;
END_VAR


VAR PERSISTENT
    //==============================================================
    // PERSISTENT — TUNING / ADJUSTMENTS
    //==============================================================
    instTUNE2_GroupSpeedDiference   : TUNE2;       // EN: XXX: "Diference" → Manual tuning helper for group speed difference / PT: XXX: "Diference" → Auxiliar de ajuste manual da diferença de velocidade do grupo
END_VAR

// ─────────────────────────────────────────────────────────────────────────────
// MAIN CALL SEQUENCE
// ─────────────────────────────────────────────────────────────────────────────
_FeedbackDisplay();
_GroupControl();          // 1) State machine: edges, enables, stop modes
_ReferenceGenerator();    // 2) Build master/slave references with ramp
_TorqueReference();       // 3) Legacy torque transfer (kept)
_StateDisplay();

_SpeedDifferenceCheck();  // 4) Speed difference monitor & trip
_alarmsDisplay();

_auxiliaryControls();

_SteamPressureControl();

_CalculateTheGearRatios();

METHOD _alarmsDisplay
VAR_INPUT
END_VAR
(*CASE groupNumber OF

    //==============================================================
    // DRYING SECTION GROUP 1 (GR1)
    //==============================================================
    1:
        //----------------------------
        // DRIVES — UPPER (GR1)
        //----------------------------
        hmiAlarms.dryingSectionGroup1UpperMasterFaultAlarm := upperMasterVfdFaultFeedback;
        hmiAlarms.dryingSectionGroup1UpperSlave1FaultAlarm := upperSlave1VfdFaultFeedback;
        hmiAlarms.dryingSectionGroup1UpperSlave2FaultAlarm := upperSlave2VfdFaultFeedback;

        //----------------------------
        // COOLING MOTORS — UPPER (GR1)
        //----------------------------
        hmiAlarms.dryingSectionGroup1UpperMasterCoolingFaultAlarm := upperMasterCoolingMotorFault;
        hmiAlarms.dryingSectionGroup1UpperSlave1CoolingFaultAlarm := upperSlave1CoolingMotorFault;
        hmiAlarms.dryingSectionGroup1UpperSlave2CoolingFaultAlarm := upperSlave2CoolingMotorFault;

        //----------------------------
        // DRIVES — LOWER (GR1)
        //----------------------------
        hmiAlarms.dryingSectionGroup1LowerMasterFaultAlarm := lowerMasterVfdFaultFeedback;
        hmiAlarms.dryingSectionGroup1LowerSlave1FaultAlarm := lowerSlave1VfdFaultFeedback;
        hmiAlarms.dryingSectionGroup1LowerSlave2FaultAlarm := lowerSlave2VfdFaultFeedback;

        //----------------------------
        // COOLING MOTORS — LOWER (GR1)
        //----------------------------
        hmiAlarms.dryingSectionGroup1LowerMasterCoolingFaultAlarm := lowerMasterCoolingMotorFault;
        hmiAlarms.dryingSectionGroup1LowerSlave1CoolingFaultAlarm := lowerSlave1CoolingMotorFault;
        hmiAlarms.dryingSectionGroup1LowerSlave2CoolingFaultAlarm := lowerSlave2CoolingMotorFault;

        //----------------------------
        // FABRIC OVERRUN SENSORS (GR1)
        //----------------------------
        hmiAlarms.upperDryingSectionGroup1FabricOverrunOperatorSideAlarm := upperDryingSectionFabricOverrunOperatorSideSensor;
        hmiAlarms.upperDryingSectionGroup1FabricOverrunDriveSideAlarm    := upperDryingSectionFabricOverrunDriveSideSensor;
        hmiAlarms.lowerDryingSectionGroup1FabricOverrunOperatorSideAlarm := lowerDryingSectionFabricOverrunOperatorSideSensor; // corrigido
        hmiAlarms.lowerDryingSectionGroup1FabricOverrunDriveSideAlarm    := lowerDryingSectionFabricOverrunDriveSideSensor;    // corrigido

        //----------------------------
        // FABRIC STRETCHER MOTOR FAULTS (GR1)
        //----------------------------
        hmiAlarms.upperDryingSectionGroup1FabricStretcherMotorFaultAlarm := upperDryingSectionFabricStretcherMotorFault;
        hmiAlarms.lowerDryingSectionGroup1FabricStretcherMotorFaultAlarm := lowerDryingSectionFabricStretcherMotorFault;


    //==============================================================
    // DRYING SECTION GROUP 2 (GR2)
    //==============================================================
    2:
        //----------------------------
        // DRIVES — UPPER (GR2)
        //----------------------------
        hmiAlarms.dryingSectionGroup2UpperMasterFaultAlarm := upperMasterVfdFaultFeedback;
        hmiAlarms.dryingSectionGroup2UpperSlave1FaultAlarm := upperSlave1VfdFaultFeedback;
        hmiAlarms.dryingSectionGroup2UpperSlave2FaultAlarm := upperSlave2VfdFaultFeedback;

        //----------------------------
        // COOLING MOTORS — UPPER (GR2)
        //----------------------------
        hmiAlarms.dryingSectionGroup2UpperMasterCoolingFaultAlarm := upperMasterCoolingMotorFault;
        hmiAlarms.dryingSectionGroup2UpperSlave1CoolingFaultAlarm := upperSlave1CoolingMotorFault;
        hmiAlarms.dryingSectionGroup2UpperSlave2CoolingFaultAlarm := upperSlave2CoolingMotorFault;

        //----------------------------
        // DRIVES — LOWER (GR2)
        //----------------------------
        hmiAlarms.dryingSectionGroup2LowerMasterFaultAlarm := lowerMasterVfdFaultFeedback;
        hmiAlarms.dryingSectionGroup2LowerSlave1FaultAlarm := lowerSlave1VfdFaultFeedback;
        hmiAlarms.dryingSectionGroup2LowerSlave2FaultAlarm := lowerSlave2VfdFaultFeedback;

        //----------------------------
        // COOLING MOTORS — LOWER (GR2)
        //----------------------------
        hmiAlarms.dryingSectionGroup2LowerMasterCoolingFaultAlarm := lowerMasterCoolingMotorFault;
        hmiAlarms.dryingSectionGroup2LowerSlave1CoolingFaultAlarm := lowerSlave1CoolingMotorFault;
        hmiAlarms.dryingSectionGroup2LowerSlave2CoolingFaultAlarm := lowerSlave2CoolingMotorFault;

        //----------------------------
        // FABRIC OVERRUN SENSORS (GR2)
        //----------------------------
        hmiAlarms.upperDryingSectionGroup2FabricOverrunOperatorSideAlarm := upperDryingSectionFabricOverrunOperatorSideSensor;
        hmiAlarms.upperDryingSectionGroup2FabricOverrunDriveSideAlarm    := upperDryingSectionFabricOverrunDriveSideSensor;
        hmiAlarms.lowerDryingSectionGroup2FabricOverrunOperatorSideAlarm := lowerDryingSectionFabricOverrunOperatorSideSensor;
        hmiAlarms.lowerDryingSectionGroup2FabricOverrunDriveSideAlarm    := lowerDryingSectionFabricOverrunDriveSideSensor;

        //----------------------------
        // FABRIC STRETCHER MOTOR FAULTS (GR2)
        //----------------------------
        hmiAlarms.upperDryingSectionGroup2FabricStretcherMotorFaultAlarm := upperDryingSectionFabricStretcherMotorFault;
        hmiAlarms.lowerDryingSectionGroup2FabricStretcherMotorFaultAlarm := lowerDryingSectionFabricStretcherMotorFault;


    //==============================================================
    // DRYING SECTION GROUP 3 (GR3)
    //==============================================================
    3:
        //----------------------------
        // DRIVES — UPPER (GR3)
        //----------------------------
        hmiAlarms.dryingSectionGroup3UpperMasterFaultAlarm := upperMasterVfdFaultFeedback;
        hmiAlarms.dryingSectionGroup3UpperSlave1FaultAlarm := upperSlave1VfdFaultFeedback;
        hmiAlarms.dryingSectionGroup3UpperSlave2FaultAlarm := upperSlave2VfdFaultFeedback;

        //----------------------------
        // COOLING MOTORS — UPPER (GR3)
        //----------------------------
        hmiAlarms.dryingSectionGroup3UpperMasterCoolingFaultAlarm := upperMasterCoolingMotorFault;
        hmiAlarms.dryingSectionGroup3UpperSlave1CoolingFaultAlarm := upperSlave1CoolingMotorFault;
        hmiAlarms.dryingSectionGroup3UpperSlave2CoolingFaultAlarm := upperSlave2CoolingMotorFault;

        //----------------------------
        // DRIVES — LOWER (GR3)
        //----------------------------
        hmiAlarms.dryingSectionGroup3LowerMasterFaultAlarm := lowerMasterVfdFaultFeedback;
        hmiAlarms.dryingSectionGroup3LowerSlave1FaultAlarm := lowerSlave1VfdFaultFeedback;
        hmiAlarms.dryingSectionGroup3LowerSlave2FaultAlarm := lowerSlave2VfdFaultFeedback;

        //----------------------------
        // COOLING MOTORS — LOWER (GR3)
        //----------------------------
        hmiAlarms.dryingSectionGroup3LowerMasterCoolingFaultAlarm := lowerMasterCoolingMotorFault;
        hmiAlarms.dryingSectionGroup3LowerSlave1CoolingFaultAlarm := lowerSlave1CoolingMotorFault;
        hmiAlarms.dryingSectionGroup3LowerSlave2CoolingFaultAlarm := lowerSlave2CoolingMotorFault;

        //----------------------------
        // FABRIC OVERRUN SENSORS (GR3)
        //----------------------------
        hmiAlarms.upperDryingSectionGroup3FabricOverrunOperatorSideAlarm := upperDryingSectionFabricOverrunOperatorSideSensor;
        hmiAlarms.upperDryingSectionGroup3FabricOverrunDriveSideAlarm    := upperDryingSectionFabricOverrunDriveSideSensor;
        hmiAlarms.lowerDryingSectionGroup3FabricOverrunOperatorSideAlarm := lowerDryingSectionFabricOverrunOperatorSideSensor;
        hmiAlarms.lowerDryingSectionGroup3FabricOverrunDriveSideAlarm    := lowerDryingSectionFabricOverrunDriveSideSensor;

        //----------------------------
        // FABRIC STRETCHER MOTOR FAULTS (GR3)
        //----------------------------
        hmiAlarms.upperDryingSectionGroup3FabricStretcherMotorFaultAlarm := upperDryingSectionFabricStretcherMotorFault;
        hmiAlarms.lowerDryingSectionGroup3FabricStretcherMotorFaultAlarm := lowerDryingSectionFabricStretcherMotorFault;


END_CASE;

//==============================================================
// GROUP FAULT — CURRENT GROUP (GR1..GR4)
//==============================================================
CASE groupNumber OF
    1:
        groupFault :=
            hmiAlarms.dryingSectionGroup1UpperMasterFaultAlarm OR
            hmiAlarms.dryingSectionGroup1UpperSlave1FaultAlarm OR
            hmiAlarms.dryingSectionGroup1UpperSlave2FaultAlarm OR
            hmiAlarms.dryingSectionGroup1LowerMasterFaultAlarm OR
            hmiAlarms.dryingSectionGroup1LowerSlave1FaultAlarm OR
            hmiAlarms.dryingSectionGroup1LowerSlave2FaultAlarm OR
            hmiAlarms.upperDryingSectionGroup1FabricOverrunOperatorSideAlarm OR
            hmiAlarms.upperDryingSectionGroup1FabricOverrunDriveSideAlarm OR
            hmiAlarms.lowerDryingSectionGroup1FabricOverrunOperatorSideAlarm OR
            hmiAlarms.lowerDryingSectionGroup1FabricOverrunDriveSideAlarm;

    2:
        groupFault :=
            hmiAlarms.dryingSectionGroup2UpperMasterFaultAlarm OR
            hmiAlarms.dryingSectionGroup2UpperSlave1FaultAlarm OR
            hmiAlarms.dryingSectionGroup2UpperSlave2FaultAlarm OR
            hmiAlarms.dryingSectionGroup2LowerMasterFaultAlarm OR
            hmiAlarms.dryingSectionGroup2LowerSlave1FaultAlarm OR
            hmiAlarms.dryingSectionGroup2LowerSlave2FaultAlarm OR
            hmiAlarms.upperDryingSectionGroup2FabricOverrunOperatorSideAlarm OR
            hmiAlarms.upperDryingSectionGroup2FabricOverrunDriveSideAlarm OR
            hmiAlarms.lowerDryingSectionGroup2FabricOverrunOperatorSideAlarm OR
            hmiAlarms.lowerDryingSectionGroup2FabricOverrunDriveSideAlarm;

    3:
        groupFault :=
            hmiAlarms.dryingSectionGroup3UpperMasterFaultAlarm OR
            hmiAlarms.dryingSectionGroup3UpperSlave1FaultAlarm OR
            hmiAlarms.dryingSectionGroup3UpperSlave2FaultAlarm OR
            hmiAlarms.dryingSectionGroup3LowerMasterFaultAlarm OR
            hmiAlarms.dryingSectionGroup3LowerSlave1FaultAlarm OR
            hmiAlarms.dryingSectionGroup3LowerSlave2FaultAlarm OR
            hmiAlarms.upperDryingSectionGroup3FabricOverrunOperatorSideAlarm OR
            hmiAlarms.upperDryingSectionGroup3FabricOverrunDriveSideAlarm OR
            hmiAlarms.lowerDryingSectionGroup3FabricOverrunOperatorSideAlarm OR
            hmiAlarms.lowerDryingSectionGroup3FabricOverrunDriveSideAlarm;


ELSE
    // Se groupNumber inválido, force seguro
    groupFault := TRUE;
END_CASE;
*)

CASE groupNumber OF

    //==============================================================
    // DRYING SECTION GROUP 1 (GR1)
    //==============================================================
    1:
        //----------------------------
        // DRIVES — UPPER (GR1)
        //----------------------------
        hmiAlarms.dryingSectionGroup1UpperMasterFaultAlarm := upperMasterVfdFaultFeedback;
        hmiAlarms.dryingSectionGroup1UpperSlave1FaultAlarm := upperSlave1VfdFaultFeedback;
        hmiAlarms.dryingSectionGroup1UpperSlave2FaultAlarm := upperSlave2VfdFaultFeedback;

        //----------------------------
        // COOLING MOTORS — UPPER (GR1)
        //----------------------------
        hmiAlarms.dryingSectionGroup1UpperMasterCoolingFaultAlarm := upperMasterCoolingMotorFault;
        hmiAlarms.dryingSectionGroup1UpperSlave1CoolingFaultAlarm := upperSlave1CoolingMotorFault;
        hmiAlarms.dryingSectionGroup1UpperSlave2CoolingFaultAlarm := upperSlave2CoolingMotorFault;

        //----------------------------
        // DRIVES — LOWER (GR1)
        //----------------------------
        hmiAlarms.dryingSectionGroup1LowerMasterFaultAlarm := lowerMasterVfdFaultFeedback;
        hmiAlarms.dryingSectionGroup1LowerSlave1FaultAlarm := lowerSlave1VfdFaultFeedback;
        hmiAlarms.dryingSectionGroup1LowerSlave2FaultAlarm := lowerSlave2VfdFaultFeedback;

        //----------------------------
        // COOLING MOTORS — LOWER (GR1)
        //----------------------------
        hmiAlarms.dryingSectionGroup1LowerMasterCoolingFaultAlarm := lowerMasterCoolingMotorFault;
        hmiAlarms.dryingSectionGroup1LowerSlave1CoolingFaultAlarm := lowerSlave1CoolingMotorFault;
        hmiAlarms.dryingSectionGroup1LowerSlave2CoolingFaultAlarm := lowerSlave2CoolingMotorFault;

        //----------------------------
        // FABRIC OVERRUN SENSORS (GR1)
        //----------------------------
        hmiAlarms.upperDryingSectionGroup1FabricOverrunOperatorSideAlarm := upperDryingSectionFabricOverrunOperatorSideSensor;
        hmiAlarms.upperDryingSectionGroup1FabricOverrunDriveSideAlarm    := upperDryingSectionFabricOverrunDriveSideSensor;
        hmiAlarms.lowerDryingSectionGroup1FabricOverrunOperatorSideAlarm := lowerDryingSectionFabricOverrunOperatorSideSensor;
        hmiAlarms.lowerDryingSectionGroup1FabricOverrunDriveSideAlarm    := lowerDryingSectionFabricOverrunDriveSideSensor;

        //----------------------------
        // FABRIC STRETCHER MOTOR FAULTS (GR1)
        //----------------------------
        hmiAlarms.upperDryingSectionGroup1FabricStretcherMotorFaultAlarm := upperDryingSectionFabricStretcherMotorFault;
        hmiAlarms.lowerDryingSectionGroup1FabricStretcherMotorFaultAlarm := lowerDryingSectionFabricStretcherMotorFault;

        //----------------------------
        // PICK-UP ROLL POSITIONER (GR1)
        //----------------------------
        // EN: Pick-up positioner fault / PT: Falha do posicionador do pick-up
        // XXX: criar em hmiAlarms: dryingSectionGroup1PickUpRollPosFaultAlarm
        hmiAlarms.dryingSectionGroup1PickUpRollPosFaultAlarm := pickUpRollPosFault;

        //----------------------------
        // SCRAPER OSCILLATORS (GR1)
        //----------------------------
        // EN: Babydryer scraper oscillator fault / PT: Falha do oscilador da raspa do babydryer
        // XXX: criar em hmiAlarms: dryingSectionGroup1BabyDryerScraperOscFaultAlarm
        hmiAlarms.dryingSectionGroup1BabyDryerScraperOscFaultAlarm := babyDryerScraperOscFault;

        // EN: Upper group scraper oscillator fault / PT: Falha do oscilador da raspa do grupo superior
        // XXX: criar em hmiAlarms: dryingSectionGroup1UpperScraperOscFaultAlarm
        hmiAlarms.dryingSectionGroup1UpperScraperOscFaultAlarm := upperGroupScraperOscFault;

        // EN: Lower group scraper oscillator fault / PT: Falha do oscilador da raspa do grupo inferior
        // XXX: criar em hmiAlarms: dryingSectionGroup1LowerScraperOscFaultAlarm
        hmiAlarms.dryingSectionGroup1LowerScraperOscFaultAlarm := lowerGroupScraperOscFault;



    //==============================================================
    // DRYING SECTION GROUP 2 (GR2)
    //==============================================================
    2:
        //----------------------------
        // DRIVES — UPPER (GR2)
        //----------------------------
        hmiAlarms.dryingSectionGroup2UpperMasterFaultAlarm := upperMasterVfdFaultFeedback;
        hmiAlarms.dryingSectionGroup2UpperSlave1FaultAlarm := upperSlave1VfdFaultFeedback;
        hmiAlarms.dryingSectionGroup2UpperSlave2FaultAlarm := upperSlave2VfdFaultFeedback;

        //----------------------------
        // COOLING MOTORS — UPPER (GR2)
        //----------------------------
        hmiAlarms.dryingSectionGroup2UpperMasterCoolingFaultAlarm := upperMasterCoolingMotorFault;
        hmiAlarms.dryingSectionGroup2UpperSlave1CoolingFaultAlarm := upperSlave1CoolingMotorFault;
        hmiAlarms.dryingSectionGroup2UpperSlave2CoolingFaultAlarm := upperSlave2CoolingMotorFault;

        //----------------------------
        // DRIVES — LOWER (GR2)
        //----------------------------
        hmiAlarms.dryingSectionGroup2LowerMasterFaultAlarm := lowerMasterVfdFaultFeedback;
        hmiAlarms.dryingSectionGroup2LowerSlave1FaultAlarm := lowerSlave1VfdFaultFeedback;
        hmiAlarms.dryingSectionGroup2LowerSlave2FaultAlarm := lowerSlave2VfdFaultFeedback;

        //----------------------------
        // COOLING MOTORS — LOWER (GR2)
        //----------------------------
        hmiAlarms.dryingSectionGroup2LowerMasterCoolingFaultAlarm := lowerMasterCoolingMotorFault;
        hmiAlarms.dryingSectionGroup2LowerSlave1CoolingFaultAlarm := lowerSlave1CoolingMotorFault;
        hmiAlarms.dryingSectionGroup2LowerSlave2CoolingFaultAlarm := lowerSlave2CoolingMotorFault;

        //----------------------------
        // FABRIC OVERRUN SENSORS (GR2)
        //----------------------------
        hmiAlarms.upperDryingSectionGroup2FabricOverrunOperatorSideAlarm := upperDryingSectionFabricOverrunOperatorSideSensor;
        hmiAlarms.upperDryingSectionGroup2FabricOverrunDriveSideAlarm    := upperDryingSectionFabricOverrunDriveSideSensor;
        hmiAlarms.lowerDryingSectionGroup2FabricOverrunOperatorSideAlarm := lowerDryingSectionFabricOverrunOperatorSideSensor;
        hmiAlarms.lowerDryingSectionGroup2FabricOverrunDriveSideAlarm    := lowerDryingSectionFabricOverrunDriveSideSensor;

        //----------------------------
        // FABRIC STRETCHER MOTOR FAULTS (GR2)
        //----------------------------
        hmiAlarms.upperDryingSectionGroup2FabricStretcherMotorFaultAlarm := upperDryingSectionFabricStretcherMotorFault;
        hmiAlarms.lowerDryingSectionGroup2FabricStretcherMotorFaultAlarm := lowerDryingSectionFabricStretcherMotorFault;

        //----------------------------
        // PICK-UP ROLL POSITIONER (GR2)
        //----------------------------
        // EN: Pick-up positioner fault / PT: Falha do posicionador do pick-up
        // XXX: criar em hmiAlarms: dryingSectionGroup2PickUpRollPosFaultAlarm
        hmiAlarms.dryingSectionGroup2PickUpRollPosFaultAlarm := pickUpRollPosFault;

        //----------------------------
        // SCRAPER OSCILLATORS (GR2)
        //----------------------------
        // XXX: dryingSectionGroup2BabyDryerScraperOscFaultAlarm
        hmiAlarms.dryingSectionGroup2BabyDryerScraperOscFaultAlarm := babyDryerScraperOscFault;
        // XXX: dryingSectionGroup2UpperScraperOscFaultAlarm
        hmiAlarms.dryingSectionGroup2UpperScraperOscFaultAlarm := upperGroupScraperOscFault;
        // XXX: dryingSectionGroup2LowerScraperOscFaultAlarm
        hmiAlarms.dryingSectionGroup2LowerScraperOscFaultAlarm := lowerGroupScraperOscFault;



    //==============================================================
    // DRYING SECTION GROUP 3 (GR3)
    //==============================================================
    3:
        //----------------------------
        // DRIVES — UPPER (GR3)
        //----------------------------
        hmiAlarms.dryingSectionGroup3UpperMasterFaultAlarm := upperMasterVfdFaultFeedback;
        hmiAlarms.dryingSectionGroup3UpperSlave1FaultAlarm := upperSlave1VfdFaultFeedback;
        hmiAlarms.dryingSectionGroup3UpperSlave2FaultAlarm := upperSlave2VfdFaultFeedback;

        //----------------------------
        // COOLING MOTORS — UPPER (GR3)
        //----------------------------
        hmiAlarms.dryingSectionGroup3UpperMasterCoolingFaultAlarm := upperMasterCoolingMotorFault;
        hmiAlarms.dryingSectionGroup3UpperSlave1CoolingFaultAlarm := upperSlave1CoolingMotorFault;
        hmiAlarms.dryingSectionGroup3UpperSlave2CoolingFaultAlarm := upperSlave2CoolingMotorFault;

        //----------------------------
        // DRIVES — LOWER (GR3)
        //----------------------------
        hmiAlarms.dryingSectionGroup3LowerMasterFaultAlarm := lowerMasterVfdFaultFeedback;
        hmiAlarms.dryingSectionGroup3LowerSlave1FaultAlarm := lowerSlave1VfdFaultFeedback;
        hmiAlarms.dryingSectionGroup3LowerSlave2FaultAlarm := lowerSlave2VfdFaultFeedback;

        //----------------------------
        // COOLING MOTORS — LOWER (GR3)
        //----------------------------
        hmiAlarms.dryingSectionGroup3LowerMasterCoolingFaultAlarm := lowerMasterCoolingMotorFault;
        hmiAlarms.dryingSectionGroup3LowerSlave1CoolingFaultAlarm := lowerSlave1CoolingMotorFault;
        hmiAlarms.dryingSectionGroup3LowerSlave2CoolingFaultAlarm := lowerSlave2CoolingMotorFault;

        //----------------------------
        // FABRIC OVERRUN SENSORS (GR3)
        //----------------------------
        hmiAlarms.upperDryingSectionGroup3FabricOverrunOperatorSideAlarm := upperDryingSectionFabricOverrunOperatorSideSensor;
        hmiAlarms.upperDryingSectionGroup3FabricOverrunDriveSideAlarm    := upperDryingSectionFabricOverrunDriveSideSensor;
        hmiAlarms.lowerDryingSectionGroup3FabricOverrunOperatorSideAlarm := lowerDryingSectionFabricOverrunOperatorSideSensor;
        hmiAlarms.lowerDryingSectionGroup3FabricOverrunDriveSideAlarm    := lowerDryingSectionFabricOverrunDriveSideSensor;

        //----------------------------
        // FABRIC STRETCHER MOTOR FAULTS (GR3)
        //----------------------------
        hmiAlarms.upperDryingSectionGroup3FabricStretcherMotorFaultAlarm := upperDryingSectionFabricStretcherMotorFault;
        hmiAlarms.lowerDryingSectionGroup3FabricStretcherMotorFaultAlarm := lowerDryingSectionFabricStretcherMotorFault;

        //----------------------------
        // PICK-UP ROLL POSITIONER (GR3)
        //----------------------------
        // XXX: dryingSectionGroup3PickUpRollPosFaultAlarm
        hmiAlarms.dryingSectionGroup3PickUpRollPosFaultAlarm := pickUpRollPosFault;

        //----------------------------
        // SCRAPER OSCILLATORS (GR3)
        //----------------------------
        // XXX: dryingSectionGroup3BabyDryerScraperOscFaultAlarm
        hmiAlarms.dryingSectionGroup3BabyDryerScraperOscFaultAlarm := babyDryerScraperOscFault;
        // XXX: dryingSectionGroup3UpperScraperOscFaultAlarm
        hmiAlarms.dryingSectionGroup3UpperScraperOscFaultAlarm := upperGroupScraperOscFault;
        // XXX: dryingSectionGroup3LowerScraperOscFaultAlarm
        hmiAlarms.dryingSectionGroup3LowerScraperOscFaultAlarm := lowerGroupScraperOscFault;

END_CASE;


//==============================================================
// GROUP FAULT — CURRENT GROUP (GR1..GR3)
//==============================================================
CASE groupNumber OF
    1:
        groupFault :=
            // Drives
            hmiAlarms.dryingSectionGroup1UpperMasterFaultAlarm OR
            hmiAlarms.dryingSectionGroup1UpperSlave1FaultAlarm OR
            hmiAlarms.dryingSectionGroup1UpperSlave2FaultAlarm OR
            hmiAlarms.dryingSectionGroup1LowerMasterFaultAlarm OR
            hmiAlarms.dryingSectionGroup1LowerSlave1FaultAlarm OR
            hmiAlarms.dryingSectionGroup1LowerSlave2FaultAlarm OR
            // Wire overrun
            hmiAlarms.upperDryingSectionGroup1FabricOverrunOperatorSideAlarm OR
            hmiAlarms.upperDryingSectionGroup1FabricOverrunDriveSideAlarm OR
            hmiAlarms.lowerDryingSectionGroup1FabricOverrunOperatorSideAlarm OR
            hmiAlarms.lowerDryingSectionGroup1FabricOverrunDriveSideAlarm OR
            // Fabric stretcher faults
            hmiAlarms.upperDryingSectionGroup1FabricStretcherMotorFaultAlarm OR
            hmiAlarms.lowerDryingSectionGroup1FabricStretcherMotorFaultAlarm OR
            // Pick-up pos fault
            // EN: Pick-up positioner fault should stop the group / PT: Falha do posicionador deve parar o grupo
            hmiAlarms.dryingSectionGroup1PickUpRollPosFaultAlarm OR
            // Scraper oscillators
            hmiAlarms.dryingSectionGroup1BabyDryerScraperOscFaultAlarm OR
            hmiAlarms.dryingSectionGroup1UpperScraperOscFaultAlarm OR
            hmiAlarms.dryingSectionGroup1LowerScraperOscFaultAlarm;

    2:
        groupFault :=
            hmiAlarms.dryingSectionGroup2UpperMasterFaultAlarm OR
            hmiAlarms.dryingSectionGroup2UpperSlave1FaultAlarm OR
            hmiAlarms.dryingSectionGroup2UpperSlave2FaultAlarm OR
            hmiAlarms.dryingSectionGroup2LowerMasterFaultAlarm OR
            hmiAlarms.dryingSectionGroup2LowerSlave1FaultAlarm OR
            hmiAlarms.dryingSectionGroup2LowerSlave2FaultAlarm OR
            hmiAlarms.upperDryingSectionGroup2FabricOverrunOperatorSideAlarm OR
            hmiAlarms.upperDryingSectionGroup2FabricOverrunDriveSideAlarm OR
            hmiAlarms.lowerDryingSectionGroup2FabricOverrunOperatorSideAlarm OR
            hmiAlarms.lowerDryingSectionGroup2FabricOverrunDriveSideAlarm;

    3:
        groupFault :=
            hmiAlarms.dryingSectionGroup3UpperMasterFaultAlarm OR
            hmiAlarms.dryingSectionGroup3UpperSlave1FaultAlarm OR
            hmiAlarms.dryingSectionGroup3UpperSlave2FaultAlarm OR
            hmiAlarms.dryingSectionGroup3LowerMasterFaultAlarm OR
            hmiAlarms.dryingSectionGroup3LowerSlave1FaultAlarm OR
            hmiAlarms.dryingSectionGroup3LowerSlave2FaultAlarm OR
            hmiAlarms.upperDryingSectionGroup3FabricOverrunOperatorSideAlarm OR
            hmiAlarms.upperDryingSectionGroup3FabricOverrunDriveSideAlarm OR
            hmiAlarms.lowerDryingSectionGroup3FabricOverrunOperatorSideAlarm OR
            hmiAlarms.lowerDryingSectionGroup3FabricOverrunDriveSideAlarm;

ELSE
    // EN: Invalid groupNumber → force safe / PT: groupNumber inválido → força seguro
    groupFault := TRUE;
END_CASE;
END_METHOD

METHOD _auxiliaryControls
VAR_INPUT
END_VAR
//==============================================
// DRYING SECTION FABRIC STRETCH / UNSTRETCH
//  - Upper & Lower groups
//  - Safe behavior: any overrun sensor blocks motion
//  - XXX: groupFault can also be added to block everything
//==============================================


//-----------------------------
// UPPER FABRIC STRETCHER
//-----------------------------
// EN: Block if motor fault OR any overrun (OS/DS)
//* PT: Bloqueia se falha de motor OU se detectar sobrecurso (LO/LA) */
IF NOT upperDryingSectionFabricStretcherMotorFault
   AND NOT upperDryingSectionFabricOverrunOperatorSideSensor
   AND NOT upperDryingSectionFabricOverrunDriveSideSensor THEN

    // Stretch
    IF upperDryingSectionFabricStretchCmd
       AND NOT upperDryingSectionFabricUnstretchCmd THEN
        upperDryingSectionFabricStretch := TRUE;
    ELSE
        upperDryingSectionFabricStretch := FALSE;
    END_IF;

    // Unstretch
    IF upperDryingSectionFabricUnstretchCmd
       AND NOT upperDryingSectionFabricStretchCmd THEN
        upperDryingSectionFabricUnstretch := TRUE;
    ELSE
        upperDryingSectionFabricUnstretch := FALSE;
    END_IF;
ELSE
    // Motor fault or overrun → force safe
    upperDryingSectionFabricStretch   := FALSE;
    upperDryingSectionFabricUnstretch := FALSE;
END_IF;


//-----------------------------
// LOWER FABRIC STRETCHER
//-----------------------------
// EN: Block if motor fault OR any overrun (OS/DS)
//* PT: Bloqueia se falha de motor OU se detectar sobrecurso (LO/LA) */
IF NOT lowerDryingSectionFabricStretcherMotorFault
   AND NOT lowerDryingSectionFabricOverrunOperatorSideSensor
   AND NOT lowerDryingSectionFabricOverrunDriveSideSensor THEN

    // Stretch
    IF lowerDryingSectionFabricStretchCmd
       AND NOT lowerDryingSectionFabricUnstretchCmd THEN
        lowerDryingSectionFabricStretch := TRUE;
    ELSE
        lowerDryingSectionFabricStretch := FALSE;
    END_IF;

    // Unstretch
    IF lowerDryingSectionFabricUnstretchCmd
       AND NOT lowerDryingSectionFabricStretchCmd THEN
        lowerDryingSectionFabricUnstretch := TRUE;
    ELSE
        lowerDryingSectionFabricUnstretch := FALSE;
    END_IF;
ELSE
    // Motor fault or overrun → force safe
    lowerDryingSectionFabricStretch   := FALSE;
    lowerDryingSectionFabricUnstretch := FALSE;
END_IF;



//==============================================
// PICK-UP ROLL POSITIONER
//  - Uses: pickUpRollPosCmdFwd / pickUpRollPosCmdRev
//  - Safety: fault or limit reached → stop
//  - Safety (optional): if both cmds = TRUE, stop
//==============================================
IF NOT pickUpRollPosFault THEN
    // Forward
    IF pickUpRollPosCmdFwd
       AND NOT pickUpRollPosCmdRev
       AND NOT pickUpRollPosLimitFwd THEN
        // EN: run forward / PT: avança
        pickUpRollPosRunFwd := TRUE;
    ELSE
        pickUpRollPosRunFwd := FALSE;
    END_IF;

    // Reverse
    IF pickUpRollPosCmdRev
       AND NOT pickUpRollPosCmdFwd
       AND NOT pickUpRollPosLimitRev THEN
        // EN: run reverse / PT: recua
        pickUpRollPosRunRev := TRUE;
    ELSE
        pickUpRollPosRunRev := FALSE;
    END_IF;
ELSE
    // EN: Fault → stop / PT: Falha → para
    pickUpRollPosRunFwd := FALSE;
    pickUpRollPosRunRev := FALSE;
END_IF;



//==============================================
// SCRAPER OSCILLATORS
//  - Babydryer
//  - Upper group
//  - Lower group
//  - Safety: fault → stop output
//==============================================

//-----------------------------
// BABYDRYER SCRAPER OSCILLATOR
//-----------------------------
IF NOT babyDryerScraperOscFault THEN
    // EN: run only if command is active / PT: aciona somente se houver comando
    IF babyDryerScraperOscCmd THEN
        babyDryerScraperOscRun := TRUE;
    ELSE
        babyDryerScraperOscRun := FALSE;
    END_IF;
ELSE
    // EN: fault → force off / PT: falha → força desligado
    babyDryerScraperOscRun := FALSE;
END_IF;


//-----------------------------
// UPPER GROUP SCRAPER OSCILLATOR
//-----------------------------
IF NOT upperGroupScraperOscFault THEN
    IF upperGroupScraperOscCmd AND upperMasterSpeedMPM > 0 THEN
        upperGroupScraperOscRun := TRUE;
    ELSE
        upperGroupScraperOscRun := FALSE;
    END_IF;
ELSE
    upperGroupScraperOscRun := FALSE;
END_IF;


//-----------------------------
// LOWER GROUP SCRAPER OSCILLATOR
//-----------------------------
IF NOT lowerGroupScraperOscFault AND lowerMasterSpeedMPM > 0 THEN
    IF lowerGroupScraperOscCmd THEN
        lowerGroupScraperOscRun := TRUE;
    ELSE
        lowerGroupScraperOscRun := FALSE;
    END_IF;
ELSE
    lowerGroupScraperOscRun := FALSE;
END_IF;
END_METHOD

METHOD _CalculateTheGearRatios
VAR_INPUT
END_VAR
VAR

END_VAR

//────────────────────────────────────────────────────────
// Gear Ratios — Upper Group (Reference: Upper Master)
//────────────────────────────────────────────────────────
IF upperMasterDiameter > 0.0 THEN

    upperToLowerMasterRatio := upperMasterDiameter / lowerMasterDiameter;

    upperToUpperSlave1Ratio := upperMasterDiameter / upperSlave1Diameter;
    upperToUpperSlave2Ratio := upperMasterDiameter / upperSlave2Diameter;

ELSE
    upperToLowerMasterRatio := 0.0;
    upperToUpperSlave1Ratio := 0.0;
    upperToUpperSlave2Ratio := 0.0;
END_IF

//────────────────────────────────────────────────────────
// Gear Ratios — Lower Group (Reference: Lower Master)
//────────────────────────────────────────────────────────
IF lowerMasterDiameter > 0.0 THEN

    lowerToUpperMasterRatio := lowerMasterDiameter / upperMasterDiameter;

    lowerToLowerSlave1Ratio := lowerMasterDiameter / lowerSlave1Diameter;
    lowerToLowerSlave2Ratio := lowerMasterDiameter / lowerSlave2Diameter;

ELSE
    lowerToUpperMasterRatio := 0.0;
    lowerToLowerSlave1Ratio := 0.0;
    lowerToLowerSlave2Ratio := 0.0;
END_IF
END_METHOD

METHOD _FeedbackDisplay
VAR_INPUT
END_VAR
(*


	
	upperMasterSpeedFilteredFeedback : REAL; // EN: Filtered upper master speed for HMI [m/min] / PT: Velocidade filtrada do mestre superior para HMI [m/min]
    upperSlave1SpeedFilteredFeedback : REAL; // EN: Filtered upper slave 1 speed for HMI [m/min] / PT: Velocidade filtrada do escravo 1 superior para HMI [m/min]
    upperSlave2SpeedFilteredFeedback : REAL; // EN: Filtered upper slave 2 speed for HMI [m/min] / PT: Velocidade filtrada do escravo 2 superior para HMI [m/min]
    lowerMasterSpeedFilteredFeedback : REAL; // EN: Filtered lower master speed for HMI [m/min] / PT: Velocidade filtrada do mestre inferior para HMI [m/min]
    lowerSlave1SpeedFilteredFeedback : REAL; // EN: Filtered lower slave 1 speed for HMI [m/min] / PT: Velocidade filtrada do escravo 1 inferior para HMI [m/min]
    lowerSlave2SpeedFilteredFeedback : REAL; // EN: Filtered lower slave 2 speed for HMI [m/min] / PT: Velocidade filtrada do escravo 2 inferior para HMI [m/min]

*)

// ── HMI display filters (PT1). Display-only; no control logic uses these values.

// UPPER GROUP — SPEED
instPT1_UpperMasterSpeedDisplay( in := upperMasterSpeedFeedback,  T := displayFilterTime, K := 1.0, out => upperMasterSpeedFilteredFeedback );
instPT1_UpperSlave1SpeedDisplay ( in := upperSlave1SpeedFeedback, T := displayFilterTime, K := 1.0, out => upperSlave1SpeedFilteredFeedback );
instPT1_UpperSlave2SpeedDisplay ( in := upperSlave2SpeedFeedback, T := displayFilterTime, K := 1.0, out => upperSlave2SpeedFilteredFeedback );

// UPPER GROUP — TORQUE
instPT1_UpperMasterTorqueDisplay( in := upperMasterTorqueFeedback,  T := displayFilterTime, K := 1.0, out => upperMasterTorqueFilteredDisplay );
instPT1_UpperSlave1TorqueDisplay ( in := upperSlave1TorqueFeedback, T := displayFilterTime, K := 1.0, out => upperSlave1TorqueFilteredDisplay );
instPT1_UpperSlave2TorqueDisplay ( in := upperSlave2TorqueFeedback, T := displayFilterTime, K := 1.0, out => upperSlave2TorqueFilteredDisplay );

// LOWER GROUP — SPEED
instPT1_LowerMasterSpeedDisplay( in := lowerMasterSpeedFeedback,  T := displayFilterTime, K := 1.0, out => lowerMasterSpeedFilteredFeedback );
instPT1_LowerSlave1SpeedDisplay( in := lowerSlave1SpeedFeedback, T := displayFilterTime, K := 1.0, out => lowerSlave1SpeedFilteredFeedback );
instPT1_LowerSlave2SpeedDisplay( in := lowerSlave2SpeedFeedback, T := displayFilterTime, K := 1.0, out => lowerSlave2SpeedFilteredFeedback );

// LOWER GROUP — TORQUE
instPT1_LowerMasterTorqueDisplay( in := lowerMasterTorqueFeedback,  T := displayFilterTime, K := 1.0, out => lowerMasterTorqueFilteredDisplay );
instPT1_LowerSlave1TorqueDisplay ( in := lowerSlave1TorqueFeedback, T := displayFilterTime, K := 1.0, out => lowerSlave1TorqueFilteredDisplay );
instPT1_LowerSlave2TorqueDisplay ( in := lowerSlave2TorqueFeedback, T := displayFilterTime, K := 1.0, out => lowerSlave2TorqueFilteredDisplay );


//====================================================================
// ═══ SPEED CALCULATION — CONVERT RPM TO MPM ════════════════════════
//====================================================================
// Formula: MPM = (π × Diameter_mm × RPM) / 1000

// ───── UPPER GROUP ─────
upperMasterSpeedMPM := (3.14159 * upperMasterDiameter * upperMasterSpeedFeedback) / 1000.0;
upperSlave1SpeedMPM := (3.14159 * upperSlave1Diameter * upperSlave1SpeedFeedback) / 1000.0;
upperSlave2SpeedMPM := (3.14159 * upperSlave2Diameter * upperSlave2SpeedFeedback) / 1000.0;

// ───── LOWER GROUP ─────
lowerMasterSpeedMPM := (3.14159 * lowerMasterDiameter * lowerMasterSpeedFeedback) / 1000.0;
lowerSlave1SpeedMPM := (3.14159 * lowerSlave1Diameter * lowerSlave1SpeedFeedback) / 1000.0;
lowerSlave2SpeedMPM := (3.14159 * lowerSlave2Diameter * lowerSlave2SpeedFeedback) / 1000.0;

// ───── UPPER GROUP ─────
upperMasterSpeedRPM := upperMasterSpeedFeedback;
upperSlave1SpeedRPM := upperSlave1SpeedFeedback;
upperSlave2SpeedRPM := upperSlave2SpeedFeedback;

// ───── LOWER GROUP ─────
lowerMasterSpeedRPM := lowerMasterSpeedFeedback;
lowerSlave1SpeedRPM := lowerSlave1SpeedFeedback;
lowerSlave2SpeedRPM := lowerSlave2SpeedFeedback;
END_METHOD

// ============================== Methods ==============================
// 1) GROUP CONTROL
METHOD _GroupControl
VAR_INPUT
END_VAR
VAR
    // Basic conditions
    speedsNearZero  : BOOL; // All drives ~0 speed
    refsNearZero    : BOOL; // Both masters ~0 ref
    allReady        : BOOL; // All six drives ready
    anyFault        : BOOL; // Any drive fault or external groupFault
	
END_VAR


// ── Edge detection ────────────────────────────────────────────────────────────
rStart := startGroup AND NOT startGroupOld;   // Start on pulse
rStop  := stopGroup  AND NOT stopGroupOld;    // Stop edge
startGroupOld := startGroup;
stopGroupOld  := stopGroup;

